C07207=1031.789,-57.070,-84.960,167.872,41.693,157.752
C07208=1031.783,-57.319,-84.950,167.870,41.694,157.752
C07209=1031.776,-57.569,-84.938,167.867,41.696,157.752
C07210=1031.770,-57.819,-84.925,167.864,41.697,157.752
C07211=1031.764,-58.068,-84.913,167.861,41.698,157.752
C07212=1031.758,-58.318,-84.902,167.859,41.700,157.752
C07213=1031.751,-58.567,-84.890,167.857,41.701,157.752
C07214=1031.746,-58.817,-84.878,167.854,41.702,157.752
C07215=1031.740,-59.067,-84.867,167.851,41.703,157.752
C07216=1031.733,-59.316,-84.855,167.848,41.705,157.752
C07217=1031.726,-59.566,-84.843,167.845,41.706,157.752
C07218=1031.721,-59.816,-84.830,167.842,41.707,157.752
C07219=1031.715,-60.065,-84.820,167.840,41.709,157.752
C07220=1031.708,-60.315,-84.808,167.838,41.710,157.752
C07221=1031.702,-60.564,-84.796,167.835,41.711,157.753
C07222=1031.697,-60.814,-84.784,167.832,41.712,157.753
C07223=1031.690,-61.064,-84.772,167.829,41.713,157.753
C07224=1031.683,-61.313,-84.760,167.826,41.714,157.753
C07225=1031.678,-61.563,-84.749,167.824,41.716,157.753
C07226=1031.672,-61.813,-84.737,167.821,41.717,157.753
C07227=1031.665,-62.063,-84.726,167.818,41.718,157.753
C07228=1031.659,-62.312,-84.714,167.815,41.719,157.753
C07229=1031.653,-62.561,-84.702,167.813,41.720,157.753
C07230=1031.647,-62.812,-84.690,167.811,41.722,157.753
C07231=1031.641,-63.061,-84.679,167.808,41.723,157.753
C07232=1031.635,-63.311,-84.667,167.805,41.724,157.753
C07233=1031.628,-63.560,-84.655,167.802,41.726,157.753
C07234=1031.623,-63.810,-84.644,167.799,41.727,157.753
C07235=1031.616,-64.060,-84.632,167.796,41.728,157.753
C07236=1031.610,-64.309,-84.620,167.793,41.729,157.753
C07237=1031.604,-64.559,-84.609,167.791,41.731,157.753
C07238=1031.597,-64.808,-84.597,167.789,41.732,157.753
C07239=1031.592,-65.058,-84.586,167.786,41.733,157.754
C07240=1031.586,-65.308,-84.574,167.783,41.735,157.754
C07241=1031.580,-65.557,-84.563,167.780,41.736,157.754
C07242=1031.573,-65.807,-84.551,167.778,41.737,157.754
C07243=1031.568,-66.057,-84.539,167.775,41.738,157.754
C07244=1031.562,-66.306,-84.527,167.772,41.740,157.754
C07245=1031.555,-66.556,-84.516,167.769,41.741,157.754
C07246=1031.549,-66.806,-84.505,167.766,41.742,157.754
C07247=1031.543,-67.055,-84.493,167.764,41.744,157.754
C07248=1031.538,-67.305,-84.482,167.762,41.744,157.754
C07249=1031.531,-67.555,-84.470,167.759,41.746,157.754
C07250=1031.525,-67.804,-84.459,167.756,41.747,157.754
C07251=1031.519,-68.087,-84.446,167.753,41.748,157.754
C07252=1031.512,-68.370,-84.433,167.749,41.750,157.754
C07253=1031.505,-68.652,-84.419,167.747,41.751,157.754
C07254=1031.498,-68.934,-84.406,167.744,41.752,157.754
C07255=1031.492,-69.185,-84.395,167.741,41.753,157.754
C07256=1031.486,-69.434,-84.384,167.738,41.755,157.755
C07257=1031.479,-69.684,-84.372,167.735,41.756,157.755
C07258=1031.474,-69.933,-84.361,167.732,41.757,157.755
C07259=1031.467,-70.183,-84.350,167.730,41.759,157.755
C07260=1031.462,-70.432,-84.338,167.727,41.760,157.755
C07261=1031.456,-70.682,-84.327,167.724,41.761,157.755
C07262=1031.450,-70.932,-84.316,167.721,41.762,157.755
C07263=1031.444,-71.181,-84.304,167.719,41.764,157.755
C07264=1031.438,-71.431,-84.293,167.717,41.765,157.755
C07265=1031.433,-71.681,-84.281,167.714,41.766,157.755
C07266=1031.426,-71.931,-84.270,167.711,41.767,157.755
C07267=1031.420,-72.180,-84.259,167.708,41.769,157.755
C07268=1031.414,-72.430,-84.247,167.705,41.770,157.755
C07269=1031.408,-72.680,-84.237,167.702,41.771,157.755
C07270=1031.402,-72.929,-84.225,167.700,41.773,157.755
C07271=1031.396,-73.179,-84.213,167.697,41.774,157.755
C07272=1031.391,-73.429,-84.202,167.694,41.775,157.755
C07273=1031.384,-73.679,-84.191,167.691,41.776,157.755
C07274=1031.378,-73.928,-84.179,167.689,41.778,157.755
///RCONF 1,0,0,1,0,0,0,0,0,0,0,0,0,0,0,0,0,0,0,0,0,0,0,0
C07275=1031.373,-74.177,-84.169,167.686,41.779,157.755
C07276=1031.366,-74.427,-84.157,167.684,41.780,157.756
C07277=1031.361,-74.677,-84.146,167.681,41.781,157.756
C07278=1031.354,-74.927,-84.135,167.678,41.783,157.756
C07279=1031.348,-75.177,-84.124,167.675,41.784,157.756
C07280=1031.343,-75.426,-84.113,167.672,41.785,157.756
C07281=1031.336,-75.676,-84.103,167.670,41.787,157.756
C07282=1031.330,-75.925,-84.092,167.667,41.788,157.756
C07283=1031.324,-76.176,-84.081,167.664,41.790,157.756
C07284=1031.318,-76.424,-84.069,167.661,41.791,157.756
C07285=1031.312,-76.674,-84.058,167.658,41.793,157.756
C07286=1031.305,-76.924,-84.047,167.656,41.794,157.756
C07287=1031.300,-77.174,-84.036,167.653,41.796,157.756
C07288=1031.294,-77.423,-84.025,167.650,41.797,157.756
C07289=1031.287,-77.673,-84.015,167.647,41.798,157.757
C07290=1031.281,-77.922,-84.004,167.644,41.799,157.757
C07291=1031.275,-78.172,-83.993,167.642,41.801,157.757
C07292=1031.269,-78.422,-83.982,167.639,41.802,157.757
C07293=1031.263,-78.672,-83.971,167.636,41.803,157.757
C07294=1031.258,-78.921,-83.960,167.633,41.805,157.757
C07295=1031.251,-79.171,-83.949,167.630,41.806,157.757
C07296=1031.246,-79.421,-83.938,167.628,41.808,157.757
C07297=1031.239,-79.670,-83.927,167.625,41.809,157.757
C07298=1031.233,-79.920,-83.916,167.622,41.811,157.757
C07299=1031.227,-80.170,-83.906,167.619,41.812,157.757
C07300=1031.222,-80.420,-83.895,167.617,41.814,157.757
C07301=1031.214,-80.670,-83.884,167.614,41.815,157.757
C07302=1031.209,-80.919,-83.874,167.611,41.816,157.757
C07303=1031.202,-81.168,-83.863,167.608,41.818,157.758
C07304=1031.196,-81.418,-83.852,167.606,41.820,157.758
C07305=1031.190,-81.669,-83.842,167.603,41.821,157.758
C07306=1031.184,-81.918,-83.832,167.600,41.823,157.758
C07307=1031.178,-82.167,-83.821,167.597,41.825,157.758
C07308=1031.171,-82.417,-83.810,167.594,41.826,157.758
C07309=1031.165,-82.667,-83.799,167.592,41.827,157.758
C07310=1031.160,-82.917,-83.789,167.589,41.828,157.758
C07311=1031.153,-83.166,-83.779,167.586,41.830,157.758
C07312=1031.147,-83.416,-83.767,167.582,41.832,157.758
C07313=1031.141,-83.666,-83.757,167.580,41.833,157.758
C07314=1031.135,-83.915,-83.747,167.577,41.835,157.759
C07315=1031.128,-84.199,-83.734,167.574,41.837,157.759
C07316=1031.121,-84.485,-83.722,167.570,41.839,157.759
C07317=1031.114,-84.769,-83.710,167.568,41.840,157.759
C07318=1031.107,-85.054,-83.698,167.564,41.842,157.759
C07319=1031.101,-85.303,-83.688,167.561,41.843,157.759
C07320=1031.096,-85.553,-83.678,167.558,41.845,157.759
C07321=1031.089,-85.803,-83.667,167.556,41.847,157.759
C07322=1031.083,-86.053,-83.656,167.553,41.848,157.759
C07323=1031.077,-86.303,-83.646,167.550,41.850,157.760
C07324=1031.071,-86.552,-83.636,167.547,41.851,157.760
C07325=1031.065,-86.802,-83.626,167.545,41.852,157.760
C07326=1031.059,-87.051,-83.615,167.542,41.854,157.760
C07327=1031.053,-87.302,-83.604,167.539,41.855,157.760
C07328=1031.046,-87.551,-83.595,167.536,41.857,157.760
C07329=1031.041,-87.801,-83.584,167.534,41.859,157.760
C07330=1031.035,-88.050,-83.573,167.531,41.860,157.760
C07331=1031.029,-88.300,-83.563,167.528,41.862,157.760
C07332=1031.023,-88.550,-83.552,167.525,41.863,157.760
C07333=1031.017,-88.799,-83.543,167.522,41.865,157.760
C07334=1031.010,-89.050,-83.532,167.520,41.866,157.761
C07335=1031.004,-89.299,-83.522,167.517,41.868,157.761
C07336=1030.999,-89.549,-83.511,167.514,41.869,157.761
///RCONF 1,0,0,0,0,0,0,0,0,0,0,0,0,0,0,0,0,0,0,0,0,0,0,0
C07337=1030.992,-89.798,-83.501,167.510,41.871,157.761
C07338=1030.987,-90.048,-83.491,167.508,41.873,157.761
C07339=1030.981,-90.298,-83.480,167.505,41.874,157.761
C07340=1030.975,-90.547,-83.470,167.502,41.876,157.761
C07341=1030.969,-90.797,-83.459,167.499,41.877,157.761
C07342=1030.963,-91.047,-83.450,167.496,41.878,157.761
C07343=1030.957,-91.296,-83.439,167.494,41.880,157.761
C07344=1030.951,-91.546,-83.429,167.491,41.882,157.761
C07345=1030.945,-91.796,-83.418,167.488,41.883,157.761
C07346=1030.938,-92.046,-83.409,167.485,41.885,157.762
C07347=1030.933,-92.296,-83.398,167.483,41.887,157.762
C07348=1030.926,-92.545,-83.388,167.480,41.888,157.762
C07349=1030.921,-92.795,-83.378,167.477,41.889,157.762
C07350=1030.915,-93.045,-83.368,167.475,41.891,157.762
C07351=1030.909,-93.295,-83.357,167.472,41.892,157.762
C07352=1030.903,-93.544,-83.347,167.469,41.894,157.762
C07353=1030.897,-93.794,-83.337,167.466,41.895,157.762
C07354=1030.892,-94.044,-83.327,167.463,41.897,157.762
C07355=1030.885,-94.293,-83.317,167.460,41.899,157.762
C07356=1030.880,-94.543,-83.306,167.457,41.900,157.762
C07357=1030.873,-94.793,-83.296,167.454,41.902,157.763
C07358=1030.868,-95.043,-83.286,167.451,41.903,157.763
C07359=1030.862,-95.292,-83.276,167.448,41.904,157.763
C07360=1030.856,-95.542,-83.266,167.446,41.906,157.763
C07361=1030.850,-95.792,-83.256,167.443,41.908,157.763
C07362=1030.844,-96.042,-83.246,167.440,41.909,157.763
C07363=1030.839,-96.290,-83.236,167.437,41.911,157.763
C07364=1030.833,-96.540,-83.226,167.435,41.913,157.763
C07365=1030.827,-96.790,-83.216,167.432,41.914,157.763
C07366=1030.821,-97.040,-83.205,167.429,41.915,157.763
C07367=1030.815,-97.290,-83.196,167.426,41.917,157.764
C07368=1030.810,-97.540,-83.186,167.424,41.918,157.764
C07369=1030.803,-97.789,-83.176,167.421,41.920,157.764
C07370=1030.797,-98.039,-83.166,167.417,41.922,157.764
C07371=1030.792,-98.289,-83.156,167.414,41.924,157.764
C07372=1030.785,-98.539,-83.146,167.412,41.925,157.764
C07373=1030.779,-98.788,-83.136,167.409,41.927,157.764
C07374=1030.773,-99.038,-83.127,167.406,41.929,157.764
C07375=1030.768,-99.288,-83.117,167.404,41.930,157.764
C07376=1030.761,-99.538,-83.107,167.401,41.932,157.764
C07377=1030.755,-99.787,-83.097,167.398,41.934,157.765
C07378=1030.749,-100.037,-83.087,167.394,41.936,157.765
C07379=1030.743,-100.324,-83.076,167.392,41.937,157.765
C07380=1030.736,-100.611,-83.065,167.388,41.939,157.765
C07381=1030.729,-100.898,-83.054,167.385,41.941,157.765
C07382=1030.722,-101.184,-83.043,167.382,41.943,157.765
C07383=1030.716,-101.434,-83.033,167.379,41.945,157.765
C07384=1030.710,-101.684,-83.023,167.376,41.946,157.765
C07385=1030.704,-101.934,-83.014,167.373,41.948,157.766
C07386=1030.698,-102.184,-83.004,167.371,41.950,157.766
C07387=1030.693,-102.433,-82.995,167.367,41.952,157.766
C07388=1030.686,-102.683,-82.985,167.364,41.954,157.766
C07389=1030.681,-102.933,-82.975,167.361,41.955,157.766
C07390=1030.674,-103.182,-82.965,167.359,41.956,157.766
C07391=1030.668,-103.432,-82.955,167.356,41.958,157.766
C07392=1030.662,-103.682,-82.946,167.353,41.960,157.766
C07393=1030.657,-103.931,-82.937,167.351,41.962,157.766
C07394=1030.651,-104.182,-82.927,167.348,41.964,157.767
C07395=1030.645,-104.431,-82.917,167.344,41.965,157.767
C07396=1030.639,-104.681,-82.908,167.341,41.967,157.767
C07397=1030.633,-104.931,-82.898,167.339,41.968,157.767
C07398=1030.627,-105.180,-82.889,167.336,41.970,157.767
C07399=1030.622,-105.430,-82.879,167.333,41.972,157.767
C07400=1030.616,-105.680,-82.869,167.330,41.974,157.767
C07401=1030.610,-105.930,-82.860,167.328,41.975,157.767
C07402=1030.603,-106.180,-82.850,167.325,41.977,157.767
C07403=1030.598,-106.429,-82.841,167.321,41.979,157.768
C07404=1030.592,-106.678,-82.831,167.319,41.981,157.768
C07405=1030.586,-106.929,-82.821,167.316,41.983,157.768
C07406=1030.580,-107.179,-82.812,167.313,41.984,157.768
C07407=1030.575,-107.428,-82.803,167.310,41.985,157.768
C07408=1030.569,-107.678,-82.794,167.308,41.987,157.768
C07409=1030.562,-107.928,-82.784,167.305,41.989,157.768
C07410=1030.556,-108.177,-82.775,167.301,41.991,157.768
C07411=1030.551,-108.427,-82.765,167.299,41.993,157.768
C07412=1030.545,-108.677,-82.756,167.296,41.995,157.769
C07413=1030.539,-108.927,-82.747,167.293,41.996,157.769
C07414=1030.533,-109.176,-82.738,167.290,41.998,157.769
C07415=1030.527,-109.426,-82.728,167.288,42.000,157.769
C07416=1030.521,-109.676,-82.719,167.284,42.002,157.769
C07417=1030.515,-109.926,-82.710,167.281,42.004,157.769
C07418=1030.509,-110.175,-82.700,167.279,42.005,157.769
C07419=1030.503,-110.425,-82.691,167.276,42.008,157.770
C07420=1030.497,-110.675,-82.682,167.273,42.010,157.770
C07421=1030.492,-110.924,-82.673,167.270,42.011,157.770
C07422=1030.486,-111.174,-82.663,167.267,42.013,157.770
C07423=1030.480,-111.425,-82.654,167.264,42.015,157.770
C07424=1030.474,-111.674,-82.645,167.262,42.017,157.770
C07425=1030.468,-111.923,-82.636,167.259,42.019,157.770
C07426=1030.462,-112.174,-82.627,167.256,42.020,157.770
C07427=1030.457,-112.423,-82.618,167.252,42.022,157.771
C07428=1030.450,-112.673,-82.608,167.250,42.024,157.771
C07429=1030.444,-112.923,-82.599,167.247,42.026,157.771
C07430=1030.439,-113.172,-82.590,167.244,42.028,157.771
C07431=1030.433,-113.422,-82.580,167.242,42.029,157.771
C07432=1030.427,-113.672,-82.572,167.239,42.031,157.771
C07433=1030.421,-113.922,-82.562,167.235,42.033,157.771
C07434=1030.415,-114.172,-82.554,167.233,42.035,157.771
C07435=1030.410,-114.421,-82.544,167.230,42.037,157.772
C07436=1030.404,-114.671,-82.535,167.227,42.038,157.772
C07437=1030.398,-114.920,-82.527,167.224,42.040,157.772
C07438=1030.392,-115.170,-82.517,167.222,42.042,157.772
C07439=1030.386,-115.420,-82.508,167.218,42.044,157.772
C07440=1030.380,-115.670,-82.499,167.215,42.046,157.772
C07441=1030.374,-115.920,-82.490,167.213,42.047,157.772
C07442=1030.369,-116.169,-82.481,167.210,42.050,157.772
C07443=1030.361,-116.456,-82.472,167.206,42.052,157.773
C07444=1030.355,-116.743,-82.461,167.203,42.054,157.773
C07445=1030.348,-117.028,-82.451,167.200,42.056,157.773
C07446=1030.342,-117.315,-82.441,167.196,42.058,157.773
C07447=1030.336,-117.565,-82.432,167.194,42.060,157.773
C07448=1030.330,-117.815,-82.423,167.191,42.062,157.773
C07449=1030.325,-118.064,-82.413,167.188,42.064,157.774
C07450=1030.318,-118.314,-82.405,167.185,42.066,157.774
C07451=1030.312,-118.563,-82.396,167.182,42.068,157.774
C07452=1030.306,-118.814,-82.387,167.179,42.070,157.774
C07453=1030.301,-119.064,-82.378,167.177,42.071,157.774
C07454=1030.294,-119.313,-82.370,167.174,42.073,157.774
C07455=1030.288,-119.563,-82.361,167.170,42.075,157.774
C07456=1030.283,-119.813,-82.352,167.168,42.078,157.774
C07457=1030.277,-120.063,-82.343,167.165,42.079,157.775
C07458=1030.272,-120.313,-82.334,167.162,42.081,157.775
C07459=1030.265,-120.561,-82.326,167.159,42.083,157.775
C07460=1030.260,-120.812,-82.317,167.156,42.085,157.775
C07461=1030.254,-121.061,-82.308,167.153,42.087,157.775
C07462=1030.248,-121.312,-82.300,167.151,42.089,157.775
C07463=1030.242,-121.561,-82.291,167.148,42.091,157.775
C07464=1030.236,-121.811,-82.282,167.144,42.093,157.776
C07465=1030.231,-122.061,-82.274,167.142,42.095,157.776
C07466=1030.225,-122.311,-82.264,167.139,42.096,157.776
C07467=1030.219,-122.560,-82.256,167.136,42.099,157.776
C07468=1030.213,-122.810,-82.247,167.134,42.101,157.776
C07469=1030.208,-123.060,-82.239,167.130,42.103,157.776
C07470=1030.202,-123.309,-82.230,167.127,42.104,157.776
C07471=1030.196,-123.559,-82.221,167.124,42.106,157.777
C07472=1030.190,-123.809,-82.213,167.122,42.108,157.777
C07473=1030.184,-124.059,-82.204,167.119,42.110,157.777
C07474=1030.179,-124.309,-82.196,167.116,42.112,157.777
C07475=1030.173,-124.558,-82.187,167.113,42.114,157.777
C07476=1030.167,-124.808,-82.178,167.110,42.116,157.777
C07477=1030.161,-125.058,-82.170,167.108,42.118,157.777
C07478=1030.155,-125.308,-82.161,167.104,42.120,157.778
C07479=1030.150,-125.558,-82.153,167.101,42.122,157.778
C07480=1030.144,-125.807,-82.145,167.098,42.124,157.778
C07481=1030.138,-126.058,-82.136,167.096,42.126,157.778
C07482=1030.132,-126.307,-82.128,167.092,42.128,157.778
C07483=1030.126,-126.556,-82.119,167.090,42.130,157.778
C07484=1030.121,-126.807,-82.110,167.087,42.133,157.779
C07485=1030.115,-127.056,-82.102,167.084,42.134,157.779
C07486=1030.109,-127.306,-82.093,167.082,42.136,157.779
C07487=1030.103,-127.556,-82.086,167.078,42.139,157.779
C07488=1030.097,-127.806,-82.077,167.075,42.140,157.779
C07489=1030.092,-128.055,-82.068,167.073,42.142,157.779
C07490=1030.087,-128.305,-82.059,167.070,42.143,157.779
C07491=1030.082,-128.554,-82.049,167.067,42.144,157.779
C07492=1030.080,-128.803,-82.038,167.065,42.145,157.779
C07493=1030.076,-129.053,-82.027,167.063,42.144,157.779
C07494=1030.074,-129.303,-82.016,167.059,42.144,157.779
C07495=1030.072,-129.554,-82.004,167.058,42.143,157.778
C07496=1030.071,-129.803,-81.991,167.056,42.142,157.778
C07497=1030.071,-130.053,-81.978,167.053,42.139,157.777
C07498=1030.071,-130.303,-81.964,167.051,42.137,157.777
C07499=1030.071,-130.553,-81.950,167.049,42.134,157.776
C07500=1030.073,-130.803,-81.934,167.048,42.131,157.776
C07501=1030.075,-131.053,-81.918,167.045,42.127,157.775
C07502=1030.077,-131.302,-81.902,167.044,42.123,157.774
C07503=1030.081,-131.553,-81.885,167.043,42.118,157.773
C07504=1030.085,-131.803,-81.868,167.042,42.112,157.772
C07505=1030.089,-132.053,-81.850,167.040,42.107,157.771
C07506=1030.095,-132.302,-81.831,167.039,42.101,157.770
C07507=1029.776,-132.327,-82.136,166.990,42.343,157.807
C07508=1029.771,-132.078,-82.154,166.992,42.349,157.808
C07509=1029.767,-131.828,-82.172,166.993,42.355,157.809
C07510=1029.762,-131.577,-82.190,166.994,42.360,157.811
C07511=1029.759,-131.327,-82.206,166.996,42.365,157.811
C07512=1029.756,-131.077,-82.223,166.997,42.369,157.812
C07513=1029.755,-130.827,-82.238,166.999,42.373,157.813
C07514=1029.753,-130.578,-82.253,167.001,42.376,157.814
C07515=1029.752,-130.328,-82.268,167.003,42.379,157.814
C07516=1029.752,-130.078,-82.282,167.004,42.382,157.815
C07517=1029.753,-129.828,-82.295,167.007,42.383,157.815
C07518=1029.754,-129.578,-82.308,167.009,42.385,157.816
C07519=1029.755,-129.328,-82.320,167.011,42.386,157.816
C07520=1029.758,-129.079,-82.332,167.013,42.387,157.816
C07521=1029.760,-128.829,-82.343,167.016,42.386,157.816
C07522=1029.764,-128.579,-82.354,167.018,42.386,157.816
C07523=1029.769,-128.330,-82.364,167.021,42.386,157.817
C07524=1029.773,-128.080,-82.373,167.024,42.384,157.816
C07525=1029.778,-127.830,-82.381,167.027,42.382,157.816
C07526=1029.784,-127.580,-82.390,167.029,42.380,157.816
C07527=1029.790,-127.332,-82.398,167.032,42.378,157.816
C07528=1029.795,-127.082,-82.407,167.036,42.376,157.816
C07529=1029.802,-126.832,-82.415,167.038,42.374,157.816
C07530=1029.807,-126.582,-82.424,167.041,42.372,157.816
C07531=1029.812,-126.332,-82.432,167.044,42.370,157.816
C07532=1029.819,-126.082,-82.440,167.047,42.368,157.815
C07533=1029.824,-125.833,-82.449,167.050,42.366,157.815
C07534=1029.830,-125.583,-82.457,167.053,42.364,157.815
C07535=1029.836,-125.333,-82.466,167.055,42.362,157.815
C07536=1029.841,-125.083,-82.474,167.059,42.360,157.815
C07537=1029.848,-124.833,-82.482,167.062,42.358,157.815
C07538=1029.854,-124.584,-82.492,167.064,42.355,157.814
C07539=1029.860,-124.334,-82.499,167.068,42.353,157.814
C07540=1029.865,-124.084,-82.508,167.070,42.352,157.814
C07541=1029.871,-123.834,-82.517,167.073,42.349,157.814
C07542=1029.877,-123.584,-82.526,167.076,42.347,157.814
C07543=1029.883,-123.335,-82.534,167.078,42.345,157.814
C07544=1029.888,-123.085,-82.543,167.082,42.344,157.814
C07545=1029.894,-122.835,-82.552,167.085,42.342,157.813
C07546=1029.900,-122.586,-82.559,167.087,42.339,157.813
C07547=1029.906,-122.335,-82.568,167.090,42.337,157.813
C07548=1029.911,-122.086,-82.578,167.094,42.335,157.813
C07549=1029.917,-121.836,-82.586,167.096,42.334,157.813
C07550=1029.923,-121.586,-82.594,167.099,42.331,157.813
C07551=1029.929,-121.337,-82.603,167.102,42.329,157.813
C07552=1029.935,-121.087,-82.612,167.105,42.327,157.812
C07553=1029.940,-120.837,-82.621,167.108,42.326,157.812
C07554=1029.947,-120.587,-82.629,167.110,42.323,157.812
C07555=1029.952,-120.338,-82.638,167.113,42.321,157.812
C07556=1029.958,-120.087,-82.647,167.116,42.320,157.812
C07557=1029.963,-119.838,-82.656,167.120,42.318,157.812
C07558=1029.970,-119.588,-82.665,167.122,42.316,157.812
C07559=1029.976,-119.338,-82.673,167.125,42.313,157.811
C07560=1029.981,-119.088,-82.682,167.127,42.311,157.811
C07561=1029.987,-118.839,-82.691,167.131,42.310,157.811
C07562=1029.993,-118.589,-82.700,167.134,42.308,157.811
C07563=1029.998,-118.339,-82.709,167.137,42.306,157.811
C07564=1030.005,-118.089,-82.717,167.139,42.303,157.811
C07565=1030.010,-117.840,-82.726,167.143,42.302,157.811
C07566=1030.016,-117.590,-82.735,167.145,42.300,157.810
C07567=1030.022,-117.340,-82.744,167.148,42.298,157.810
C07568=1030.029,-117.054,-82.754,167.152,42.295,157.810
C07569=1030.035,-116.768,-82.765,167.154,42.293,157.810
C07570=1030.042,-116.481,-82.774,167.158,42.292,157.810
C07571=1030.049,-116.195,-82.785,167.162,42.289,157.810
C07572=1030.055,-115.945,-82.794,167.164,42.287,157.810
C07573=1030.061,-115.695,-82.803,167.167,42.285,157.809
C07574=1030.066,-115.446,-82.812,167.170,42.284,157.809
C07575=1030.073,-115.196,-82.821,167.173,42.281,157.809
C07576=1030.078,-114.947,-82.830,167.176,42.279,157.809
C07577=1030.084,-114.696,-82.839,167.179,42.277,157.809
C07578=1030.090,-114.446,-82.848,167.181,42.275,157.809
C07579=1030.096,-114.197,-82.857,167.185,42.274,157.809
C07580=1030.102,-113.947,-82.866,167.188,42.272,157.809
C07581=1030.107,-113.697,-82.875,167.190,42.270,157.808
C07582=1030.113,-113.447,-82.884,167.193,42.268,157.808
C07583=1030.119,-113.198,-82.894,167.196,42.266,157.808
C07584=1030.125,-112.948,-82.902,167.199,42.265,157.808
C07585=1030.131,-112.698,-82.912,167.202,42.263,157.808
C07586=1030.136,-112.448,-82.920,167.205,42.260,157.808
C07587=1030.142,-112.199,-82.930,167.207,42.258,157.808
C07588=1030.148,-111.949,-82.940,167.210,42.257,157.807
C07589=1030.154,-111.699,-82.948,167.213,42.255,157.807
C07590=1030.160,-111.449,-82.958,167.217,42.253,157.807
C07591=1030.166,-111.199,-82.967,167.219,42.251,157.807
C07592=1030.171,-110.950,-82.976,167.222,42.249,157.807
C07593=1030.177,-110.700,-82.985,167.225,42.247,157.807
C07594=1030.184,-110.450,-82.995,167.227,42.246,157.807
C07595=1030.189,-110.200,-83.003,167.231,42.244,157.807
C07596=1030.195,-109.951,-83.013,167.234,42.242,157.807
C07597=1030.201,-109.701,-83.022,167.236,42.240,157.806
C07598=1030.207,-109.452,-83.032,167.239,42.238,157.806
C07599=1030.213,-109.201,-83.041,167.242,42.237,157.806
C07600=1030.219,-108.951,-83.050,167.246,42.235,157.806
C07601=1030.224,-108.702,-83.059,167.248,42.233,157.806
C07602=1030.231,-108.453,-83.069,167.251,42.230,157.806
C07603=1030.236,-108.202,-83.078,167.253,42.229,157.806
C07604=1030.243,-107.952,-83.087,167.256,42.227,157.805
C07605=1030.248,-107.703,-83.096,167.260,42.225,157.805
C07606=1030.254,-107.453,-83.106,167.263,42.223,157.805
C07607=1030.261,-107.204,-83.116,167.265,42.221,157.805
C07608=1030.266,-106.953,-83.124,167.268,42.219,157.805
C07609=1030.272,-106.704,-83.134,167.271,42.218,157.805
C07610=1030.278,-106.454,-83.143,167.273,42.216,157.805
C07611=1030.284,-106.204,-83.153,167.277,42.214,157.805
C07612=1030.290,-105.954,-83.163,167.280,42.213,157.805
C07613=1030.295,-105.705,-83.172,167.283,42.211,157.804
C07614=1030.302,-105.456,-83.182,167.285,42.209,157.804
C07615=1030.308,-105.206,-83.191,167.288,42.207,157.804
C07616=1030.314,-104.956,-83.201,167.291,42.206,157.804
C07617=1030.319,-104.705,-83.210,167.294,42.204,157.804
C07618=1030.325,-104.456,-83.220,167.297,42.202,157.804
C07619=1030.331,-104.206,-83.229,167.300,42.200,157.804
C07620=1030.337,-103.957,-83.239,167.302,42.198,157.804
C07621=1030.343,-103.707,-83.248,167.305,42.197,157.803
C07622=1030.348,-103.457,-83.258,167.308,42.195,157.803
C07623=1030.354,-103.208,-83.268,167.311,42.193,157.803
C07624=1030.360,-102.958,-83.277,167.314,42.191,157.803
C07625=1030.366,-102.708,-83.287,167.317,42.189,157.803
C07626=1030.373,-102.458,-83.296,167.320,42.188,157.803
C07627=1030.378,-102.208,-83.306,167.323,42.186,157.803
C07628=1030.384,-101.959,-83.316,167.325,42.185,157.803
C07629=1030.390,-101.709,-83.325,167.328,42.183,157.803
C07630=1030.396,-101.459,-83.335,167.332,42.181,157.803
C07631=1030.402,-101.210,-83.346,167.334,42.179,157.802
C07632=1030.408,-100.923,-83.357,167.337,42.177,157.802
C07633=1030.416,-100.636,-83.368,167.341,42.175,157.802
C07634=1030.422,-100.349,-83.379,167.344,42.173,157.802
C07635=1030.429,-100.063,-83.390,167.347,42.171,157.802
C07636=1030.435,-99.813,-83.399,167.350,42.169,157.802
C07637=1030.441,-99.563,-83.409,167.352,42.167,157.802
C07638=1030.447,-99.313,-83.419,167.356,42.165,157.802
C07639=1030.453,-99.063,-83.428,167.359,42.164,157.802
C07640=1030.460,-98.814,-83.439,167.362,42.163,157.801
C07641=1030.465,-98.564,-83.449,167.364,42.161,157.801
C07642=1030.471,-98.314,-83.458,167.367,42.159,157.801
C07643=1030.477,-98.064,-83.468,167.370,42.157,157.801
C07644=1030.483,-97.815,-83.478,167.373,42.155,157.801
C07645=1030.489,-97.564,-83.488,167.376,42.154,157.801
C07646=1030.495,-97.315,-83.498,167.379,42.152,157.801
C07647=1030.501,-97.065,-83.508,167.382,42.151,157.801
C07648=1030.506,-96.816,-83.517,167.384,42.149,157.800
C07649=1030.512,-96.566,-83.527,167.387,42.147,157.800
C07650=1030.518,-96.317,-83.538,167.390,42.146,157.800
C07651=1030.524,-96.067,-83.548,167.393,42.144,157.800
C07652=1030.530,-95.817,-83.557,167.395,42.142,157.800
C07653=1030.536,-95.567,-83.568,167.398,42.141,157.800
C07654=1030.542,-95.318,-83.578,167.401,42.140,157.800
C07655=1030.547,-95.067,-83.588,167.405,42.138,157.800
C07656=1030.554,-94.818,-83.598,167.407,42.136,157.800
C07657=1030.559,-94.568,-83.609,167.410,42.134,157.800
C07658=1030.565,-94.318,-83.618,167.413,42.133,157.800
C07659=1030.571,-94.069,-83.629,167.416,42.131,157.799
C07660=1030.577,-93.819,-83.639,167.418,42.129,157.799
C07661=1030.583,-93.570,-83.649,167.421,42.128,157.799
C07662=1030.589,-93.320,-83.659,167.424,42.127,157.799
C07663=1030.595,-93.070,-83.669,167.427,42.125,157.799
C07664=1030.601,-92.821,-83.679,167.429,42.123,157.799
C07665=1030.607,-92.570,-83.690,167.432,42.122,157.799
C07666=1030.612,-92.321,-83.700,167.436,42.120,157.799
C07667=1030.618,-92.071,-83.710,167.439,42.118,157.799
C07668=1030.624,-91.822,-83.721,167.441,42.117,157.799
C07669=1030.630,-91.572,-83.730,167.444,42.115,157.799
C07670=1030.636,-91.322,-83.741,167.447,42.113,157.798
C07671=1030.642,-91.073,-83.751,167.449,42.112,157.798
C07672=1030.648,-90.822,-83.761,167.452,42.111,157.798
C07673=1030.654,-90.573,-83.771,167.455,42.109,157.798
C07674=1030.660,-90.322,-83.782,167.458,42.107,157.798
C07675=1030.667,-90.073,-83.792,167.461,42.106,157.798
C07676=1030.672,-89.823,-83.802,167.463,42.104,157.798
C07677=1030.679,-89.574,-83.813,167.466,42.102,157.798
C07678=1030.684,-89.324,-83.824,167.470,42.100,157.798
C07679=1030.690,-89.074,-83.834,167.473,42.099,157.798
C07680=1030.696,-88.825,-83.844,167.475,42.098,157.798
C07681=1030.702,-88.575,-83.854,167.478,42.096,157.797
C07682=1030.708,-88.326,-83.864,167.481,42.095,157.797
C07683=1030.714,-88.076,-83.875,167.484,42.093,157.797
C07684=1030.721,-87.826,-83.885,167.486,42.091,157.797
C07685=1030.726,-87.576,-83.896,167.489,42.089,157.797
C07686=1030.732,-87.326,-83.906,167.492,42.088,157.797
C07687=1030.738,-87.077,-83.917,167.495,42.087,157.797
C07688=1030.744,-86.827,-83.927,167.497,42.085,157.797
C07689=1030.750,-86.578,-83.937,167.500,42.084,157.797
C07690=1030.757,-86.328,-83.948,167.503,42.082,157.797
C07691=1030.763,-86.078,-83.958,167.507,42.080,157.797
C07692=1030.768,-85.828,-83.969,167.509,42.079,157.797
C07693=1030.774,-85.579,-83.980,167.512,42.077,157.796
C07694=1030.780,-85.329,-83.989,167.515,42.075,157.796
C07695=1030.786,-85.080,-84.000,167.517,42.074,157.796
C07696=1030.793,-84.794,-84.012,167.520,42.072,157.796
C07697=1030.801,-84.510,-84.024,167.524,42.070,157.796
C07698=1030.808,-84.225,-84.036,167.527,42.069,157.796
C07699=1030.814,-83.941,-84.047,167.530,42.067,157.796
C07700=1030.820,-83.691,-84.058,167.533,42.065,157.796
C07701=1030.827,-83.442,-84.069,167.536,42.063,157.796
C07702=1030.833,-83.192,-84.080,167.539,42.062,157.795
C07703=1030.838,-82.942,-84.090,167.541,42.060,157.795
C07704=1030.845,-82.692,-84.100,167.544,42.059,157.795
C07705=1030.851,-82.443,-84.111,167.547,42.057,157.795
C07706=1030.858,-82.193,-84.122,167.550,42.056,157.795
C07707=1030.863,-81.943,-84.132,167.552,42.054,157.795
C07708=1030.869,-81.694,-84.143,167.556,42.052,157.795
C07709=1030.876,-81.444,-84.154,167.559,42.050,157.795
C07710=1030.882,-81.194,-84.164,167.562,42.049,157.795
C07711=1030.888,-80.945,-84.175,167.564,42.047,157.795
C07712=1030.894,-80.695,-84.185,167.567,42.046,157.794
C07713=1030.900,-80.445,-84.196,167.570,42.045,157.794
C07714=1030.906,-80.195,-84.206,167.573,42.043,157.794
C07715=1030.912,-79.946,-84.217,167.575,42.041,157.794
C07716=1030.918,-79.696,-84.229,167.578,42.040,157.794
C07717=1030.924,-79.446,-84.239,167.581,42.038,157.794
C07718=1030.931,-79.197,-84.250,167.584,42.037,157.794
C07719=1030.937,-78.947,-84.261,167.586,42.035,157.794
C07720=1030.943,-78.697,-84.272,167.589,42.034,157.794
C07721=1030.948,-78.448,-84.283,167.592,42.032,157.794
C07722=1030.955,-78.198,-84.294,167.595,42.031,157.794
C07723=1030.961,-77.948,-84.305,167.598,42.030,157.794
C07724=1030.966,-77.699,-84.316,167.600,42.028,157.793
C07725=1030.973,-77.449,-84.327,167.603,42.027,157.793
C07726=1030.979,-77.199,-84.337,167.606,42.025,157.793
C07727=1030.985,-76.950,-84.348,167.609,42.024,157.793
C07728=1030.991,-76.700,-84.359,167.611,42.022,157.793
C07729=1030.997,-76.450,-84.370,167.614,42.021,157.793
C07730=1031.003,-76.201,-84.381,167.617,42.019,157.793
C07731=1031.009,-75.951,-84.392,167.620,42.018,157.793
C07732=1031.015,-75.701,-84.403,167.623,42.016,157.793
C07733=1031.020,-75.452,-84.414,167.625,42.015,157.793
C07734=1031.028,-75.202,-84.425,167.628,42.014,157.793
C07735=1031.033,-74.952,-84.436,167.631,42.012,157.793
C07736=1031.040,-74.702,-84.447,167.634,42.011,157.793
C07737=1031.045,-74.453,-84.458,167.637,42.010,157.793
C07738=1031.051,-74.203,-84.469,167.639,42.008,157.792
C07739=1031.058,-73.953,-84.481,167.642,42.007,157.792
C07740=1031.064,-73.704,-84.491,167.645,42.005,157.792
///RCONF 1,0,0,1,0,0,0,0,0,0,0,0,0,0,0,0,0,0,0,0,0,0,0,0
C07741=1031.070,-73.454,-84.503,167.648,42.004,157.792
C07742=1031.075,-73.204,-84.514,167.651,42.003,157.792
C07743=1031.081,-72.955,-84.525,167.653,42.001,157.792
C07744=1031.087,-72.705,-84.537,167.656,42.000,157.792
C07745=1031.093,-72.455,-84.548,167.659,41.999,157.792
C07746=1031.099,-72.205,-84.559,167.662,41.997,157.792
C07747=1031.105,-71.956,-84.570,167.665,41.996,157.792
C07748=1031.110,-71.707,-84.582,167.668,41.995,157.792
C07749=1031.117,-71.456,-84.593,167.670,41.993,157.792
C07750=1031.122,-71.207,-84.604,167.672,41.992,157.792
C07751=1031.129,-70.957,-84.616,167.675,41.991,157.792
C07752=1031.135,-70.708,-84.627,167.678,41.989,157.792
C07753=1031.141,-70.458,-84.638,167.681,41.988,157.792
C07754=1031.146,-70.208,-84.651,167.683,41.987,157.792
C07755=1031.153,-69.958,-84.662,167.686,41.985,157.791
C07756=1031.159,-69.709,-84.673,167.689,41.984,157.791
C07757=1031.165,-69.460,-84.684,167.692,41.983,157.791
C07758=1031.171,-69.210,-84.696,167.695,41.981,157.791
C07759=1031.176,-68.960,-84.707,167.697,41.980,157.791
C07760=1031.183,-68.678,-84.719,167.700,41.979,157.791
C07761=1031.190,-68.395,-84.732,167.703,41.978,157.791
C07762=1031.197,-68.113,-84.746,167.707,41.976,157.791
C07763=1031.204,-67.830,-84.759,167.710,41.975,157.791
C07764=1031.210,-67.580,-84.770,167.712,41.973,157.791
C07765=1031.216,-67.330,-84.781,167.715,41.972,157.791
C07766=1031.222,-67.081,-84.794,167.718,41.971,157.791
C07767=1031.228,-66.831,-84.805,167.721,41.969,157.791
C07768=1031.234,-66.582,-84.817,167.724,41.968,157.791
C07769=1031.240,-66.332,-84.828,167.726,41.967,157.791
C07770=1031.247,-66.082,-84.839,167.729,41.965,157.791
C07771=1031.252,-65.833,-84.851,167.732,41.964,157.791
C07772=1031.258,-65.583,-84.863,167.734,41.963,157.791
C07773=1031.265,-65.333,-84.874,167.737,41.961,157.790
C07774=1031.271,-65.084,-84.886,167.739,41.960,157.790
C07775=1031.277,-64.834,-84.897,167.742,41.959,157.790
C07776=1031.282,-64.585,-84.909,167.745,41.957,157.790
C07777=1031.289,-64.334,-84.920,167.748,41.956,157.790
C07778=1031.295,-64.086,-84.932,167.751,41.954,157.790
C07779=1031.301,-63.835,-84.943,167.753,41.953,157.790
C07780=1031.307,-63.586,-84.956,167.756,41.952,157.790
C07781=1031.313,-63.336,-84.967,167.759,41.950,157.790
C07782=1031.319,-63.086,-84.979,167.762,41.949,157.790
C07783=1031.326,-62.836,-84.990,167.765,41.948,157.790
C07784=1031.331,-62.587,-85.002,167.766,41.947,157.790
C07785=1031.338,-62.338,-85.014,167.769,41.946,157.790
C07786=1031.343,-62.088,-85.025,167.772,41.944,157.790
C07787=1031.350,-61.838,-85.037,167.775,41.943,157.790
C07788=1031.356,-61.588,-85.048,167.778,41.942,157.790
C07789=1031.362,-61.339,-85.060,167.781,41.941,157.790
C07790=1031.368,-61.090,-85.072,167.783,41.939,157.789
C07791=1031.375,-60.839,-85.083,167.786,41.938,157.789
C07792=1031.381,-60.590,-85.095,167.789,41.936,157.789
C07793=1031.387,-60.341,-85.108,167.792,41.935,157.789
C07794=1031.393,-60.090,-85.119,167.795,41.934,157.789
C07795=1031.399,-59.842,-85.130,167.797,41.932,157.789
C07796=1031.406,-59.592,-85.142,167.799,41.931,157.789
C07797=1031.411,-59.341,-85.154,167.802,41.930,157.789
C07798=1031.418,-59.092,-85.166,167.805,41.928,157.789
C07799=1031.424,-58.843,-85.178,167.808,41.927,157.789
C07800=1031.430,-58.593,-85.189,167.811,41.926,157.789
C07801=1031.436,-58.343,-85.202,167.813,41.924,157.789
C07802=1031.443,-58.093,-85.214,167.816,41.923,157.789
C07803=1031.449,-57.844,-85.225,167.819,41.922,157.789
C07804=1031.455,-57.594,-85.237,167.822,41.920,157.789
C07805=1031.461,-57.344,-85.249,167.825,41.919,157.789
C07806=1031.468,-57.095,-85.261,167.827,41.918,157.788
C07807=1031.474,-56.846,-85.273,167.829,41.917,157.788
///RCONF 1,0,0,0,0,0,0,0,0,0,0,0,0,0,0,0,0,0,0,0,0,0,0,0
C07808=1031.480,-56.595,-85.284,167.832,41.915,157.788
C07809=1031.486,-56.346,-85.296,167.835,41.914,157.788
C07810=1031.493,-56.096,-85.308,167.838,41.913,157.788
C07811=1031.499,-55.847,-85.320,167.840,41.912,157.788
C07812=1031.505,-55.598,-85.332,167.843,41.910,157.788
C07813=1031.511,-55.347,-85.344,167.846,41.909,157.788
C07814=1031.518,-55.098,-85.356,167.849,41.907,157.788
C07815=1031.524,-54.848,-85.368,167.852,41.906,157.788
C07816=1031.530,-54.599,-85.380,167.854,41.905,157.788
C07817=1031.536,-54.349,-85.392,167.856,41.903,157.788
C07818=1031.543,-54.100,-85.404,167.859,41.902,157.788
C07819=1031.549,-53.849,-85.416,167.862,41.901,157.788
C07820=1031.555,-53.600,-85.427,167.865,41.899,157.787
C07821=1031.562,-53.350,-85.439,167.867,41.898,157.787
C07822=1031.567,-53.101,-85.452,167.870,41.896,157.787
C07823=1031.574,-52.852,-85.464,167.873,41.895,157.787
C07824=1031.581,-52.569,-85.477,167.876,41.894,157.787
C07825=1031.588,-52.289,-85.491,167.879,41.893,157.787
C07826=1031.595,-52.007,-85.504,167.882,41.891,157.787
C07827=1031.603,-51.727,-85.518,167.885,41.890,157.787
C07828=1031.609,-51.477,-85.531,167.888,41.888,157.787
C07829=1031.615,-51.227,-85.542,167.891,41.887,157.787
C07830=1031.622,-50.978,-85.554,167.894,41.886,157.787
C07831=1031.628,-50.727,-85.566,167.895,41.884,157.787
C07832=1031.634,-50.478,-85.578,167.898,41.883,157.787
C07833=1031.640,-50.229,-85.591,167.901,41.882,157.787
C07834=1031.647,-49.979,-85.603,167.904,41.881,157.787
C07835=1031.653,-49.730,-85.616,167.907,41.880,157.787
C07836=1031.658,-49.480,-85.628,167.909,41.879,157.787
C07837=1031.664,-49.230,-85.641,167.911,41.877,157.786
C07838=1031.671,-48.980,-85.653,167.914,41.876,157.786
C07839=1031.677,-48.730,-85.665,167.917,41.875,157.786
C07840=1031.683,-48.480,-85.678,167.920,41.874,157.786
C07841=1031.689,-48.232,-85.689,167.923,41.873,157.786
C07842=1031.695,-47.982,-85.703,167.925,41.872,157.786
C07843=1031.701,-47.732,-85.715,167.928,41.871,157.786
C07844=1031.708,-47.483,-85.727,167.930,41.869,157.786
C07845=1031.714,-47.233,-85.740,167.933,41.868,157.786
C07846=1031.719,-46.983,-85.752,167.936,41.867,157.786
C07847=1031.726,-46.733,-85.764,167.938,41.866,157.786
C07848=1031.732,-46.484,-85.778,167.941,41.865,157.786
C07849=1031.738,-46.234,-85.790,167.944,41.864,157.786
C07850=1031.745,-45.985,-85.802,167.947,41.863,157.786
C07851=1031.751,-45.735,-85.815,167.949,41.861,157.786
C07852=1031.757,-45.486,-85.828,167.951,41.860,157.786
C07853=1031.764,-45.236,-85.840,167.954,41.859,157.786
C07854=1031.770,-44.986,-85.852,167.957,41.858,157.786
C07855=1031.775,-44.736,-85.865,167.960,41.857,157.786
C07856=1031.782,-44.487,-85.878,167.962,41.856,157.786
C07857=1031.788,-44.237,-85.890,167.964,41.855,157.786
C07858=1031.794,-43.988,-85.903,167.967,41.853,157.786
C07859=1031.800,-43.738,-85.915,167.970,41.852,157.786
C07860=1031.807,-43.489,-85.928,167.973,41.851,157.786
C07861=1031.813,-43.239,-85.941,167.975,41.850,157.786
C07862=1031.819,-42.989,-85.953,167.978,41.849,157.786
C07863=1031.826,-42.740,-85.966,167.980,41.848,157.785
C07864=1031.832,-42.490,-85.978,167.983,41.847,157.785
C07865=1031.838,-42.240,-85.991,167.986,41.845,157.785
C07866=1031.844,-41.991,-86.004,167.988,41.844,157.785
C07867=1031.851,-41.741,-86.016,167.991,41.843,157.785
C07868=1031.857,-41.492,-86.029,167.994,41.842,157.785
C07869=1031.863,-41.242,-86.042,167.997,41.841,157.785
C07870=1031.869,-40.993,-86.054,167.999,41.840,157.785
C07871=1031.876,-40.743,-86.067,168.001,41.838,157.785
C07872=1031.881,-40.494,-86.080,168.004,41.837,157.785
C07873=1031.887,-40.244,-86.092,168.007,41.836,157.785
C07874=1031.894,-39.995,-86.105,168.010,41.835,157.785
C07875=1031.900,-39.745,-86.117,168.012,41.834,157.785
C07876=1031.906,-39.496,-86.131,168.014,41.833,157.785
C07877=1031.912,-39.246,-86.143,168.017,41.831,157.785
C07878=1031.919,-38.997,-86.156,168.020,41.830,157.785
C07879=1031.926,-38.746,-86.169,168.023,41.829,157.785
C07880=1031.932,-38.497,-86.182,168.025,41.828,157.785
C07881=1031.938,-38.247,-86.195,168.028,41.827,157.785
C07882=1031.944,-37.998,-86.208,168.030,41.826,157.785
C07883=1031.950,-37.748,-86.221,168.032,41.825,157.785
C07884=1031.956,-37.499,-86.234,168.035,41.824,157.785
C07885=1031.962,-37.249,-86.246,168.038,41.823,157.785
C07886=1031.968,-36.999,-86.260,168.041,41.822,157.785
C07887=1031.975,-36.750,-86.273,168.043,41.821,157.784
C07888=1031.982,-36.469,-86.287,168.046,41.820,157.784
C07889=1031.989,-36.188,-86.301,168.049,41.819,157.784
C07890=1031.995,-35.908,-86.317,168.051,41.817,157.784
C07891=1032.002,-35.626,-86.331,168.055,41.816,157.784
C07892=1032.009,-35.377,-86.344,168.057,41.815,157.784
C07893=1032.015,-35.128,-86.358,168.060,41.814,157.784
C07894=1032.021,-34.878,-86.370,168.063,41.813,157.784
C07895=1032.027,-34.629,-86.384,168.065,41.812,157.784
C07896=1032.034,-34.379,-86.397,168.067,41.811,157.784
C07897=1032.040,-34.129,-86.410,168.070,41.809,157.784
C07898=1032.046,-33.879,-86.423,168.073,41.808,157.784
C07899=1032.052,-33.630,-86.436,168.075,41.807,157.784
C07900=1032.058,-33.380,-86.449,168.078,41.806,157.784
C07901=1032.064,-33.131,-86.462,168.081,41.805,157.784
C07902=1032.071,-32.881,-86.476,168.083,41.804,157.784
C07903=1032.077,-32.631,-86.488,168.086,41.803,157.784
C07904=1032.083,-32.382,-86.502,168.088,41.802,157.784
C07905=1032.089,-32.133,-86.515,168.091,41.801,157.784
C07906=1032.096,-31.883,-86.528,168.093,41.800,157.784
C07907=1032.102,-31.633,-86.541,168.096,41.799,157.784
C07908=1032.108,-31.384,-86.554,168.099,41.798,157.784
C07909=1032.115,-31.134,-86.568,168.101,41.797,157.784
C07910=1032.121,-30.885,-86.581,168.104,41.796,157.784
C07911=1032.127,-30.634,-86.594,168.107,41.795,157.784
C07912=1032.133,-30.385,-86.607,168.108,41.794,157.784
C07913=1032.140,-30.136,-86.620,168.111,41.793,157.784
C07914=1032.146,-29.887,-86.634,168.114,41.792,157.784
C07915=1032.153,-29.637,-86.647,168.117,41.791,157.784
C07916=1032.159,-29.387,-86.660,168.119,41.790,157.784
C07917=1032.165,-29.138,-86.673,168.122,41.788,157.783
C07918=1032.171,-28.888,-86.686,168.124,41.787,157.783
C07919=1032.178,-28.638,-86.700,168.126,41.786,157.783
C07920=1032.184,-28.389,-86.713,168.129,41.785,157.783
C07921=1032.190,-28.140,-86.726,168.132,41.784,157.783
C07922=1032.197,-27.890,-86.740,168.135,41.783,157.783
C07923=1032.203,-27.640,-86.753,168.137,41.782,157.783
C07924=1032.209,-27.391,-86.766,168.140,41.781,157.783
C07925=1032.215,-27.141,-86.779,168.142,41.780,157.783
C07926=1032.221,-26.891,-86.793,168.144,41.779,157.783
C07927=1032.228,-26.642,-86.807,168.147,41.778,157.783
C07928=1032.234,-26.393,-86.820,168.150,41.777,157.783
C07929=1032.240,-26.142,-86.834,168.152,41.776,157.783
C07930=1032.246,-25.893,-86.847,168.155,41.775,157.783
C07931=1032.252,-25.644,-86.861,168.157,41.775,157.783
C07932=1032.259,-25.393,-86.875,168.160,41.773,157.783
C07933=1032.265,-25.144,-86.888,168.163,41.772,157.783
C07934=1032.271,-24.895,-86.901,168.164,41.771,157.783
C07935=1032.277,-24.646,-86.915,168.167,41.770,157.783
C07936=1032.283,-24.395,-86.929,168.170,41.769,157.783
C07937=1032.289,-24.146,-86.942,168.172,41.768,157.783
C07938=1032.296,-23.897,-86.956,168.175,41.767,157.783
C07939=1032.302,-23.647,-86.970,168.178,41.766,157.783
C07940=1032.308,-23.398,-86.984,168.180,41.765,157.783
C07941=1032.314,-23.149,-86.997,168.183,41.765,157.783
C07942=1032.321,-22.899,-87.011,168.185,41.764,157.783
C07943=1032.327,-22.649,-87.025,168.187,41.763,157.783
C07944=1032.334,-22.334,-87.042,168.190,41.762,157.783
C07945=1032.343,-22.019,-87.059,168.194,41.760,157.783
C07946=1032.351,-21.704,-87.076,168.197,41.759,157.783
C07947=1032.359,-21.389,-87.093,168.200,41.758,157.783
C07948=1032.364,-21.156,-87.106,168.203,41.757,157.783
C07949=1032.370,-20.923,-87.119,168.204,41.756,157.783
C07950=1032.376,-20.690,-87.132,168.207,41.755,157.783
C07951=1032.382,-20.458,-87.145,168.209,41.754,157.783
C07952=1032.388,-20.225,-87.158,168.212,41.753,157.783
C07953=1032.394,-19.992,-87.171,168.214,41.752,157.783
C07954=1032.400,-19.759,-87.183,168.217,41.751,157.783
C07955=1032.405,-19.526,-87.196,168.219,41.750,157.783
C07956=1032.412,-19.277,-87.209,168.222,41.749,157.783
C07957=1032.418,-19.027,-87.224,168.224,41.748,157.782
C07958=1032.424,-18.778,-87.237,168.226,41.747,157.782
C07959=1032.431,-18.528,-87.251,168.228,41.746,157.782
C07960=1032.436,-18.278,-87.265,168.231,41.745,157.782
C07961=1032.443,-18.029,-87.279,168.234,41.744,157.782
C07962=1032.450,-17.780,-87.293,168.236,41.743,157.782
C07963=1032.455,-17.530,-87.306,168.239,41.742,157.782
C07964=1032.462,-17.280,-87.320,168.242,41.742,157.782
C07965=1032.469,-17.031,-87.334,168.244,41.741,157.782
C07966=1032.475,-16.781,-87.348,168.247,41.740,157.782
C07967=1032.481,-16.532,-87.362,168.248,41.739,157.782
C07968=1032.488,-16.282,-87.376,168.251,41.738,157.782
C07969=1032.494,-16.033,-87.390,168.254,41.737,157.782
C07970=1032.500,-15.783,-87.403,168.256,41.736,157.782
C07971=1032.507,-15.534,-87.417,168.259,41.735,157.782
C07972=1032.513,-15.284,-87.432,168.261,41.734,157.782
C07973=1032.519,-15.035,-87.445,168.264,41.733,157.782
C07974=1032.526,-14.785,-87.460,168.266,41.732,157.782
C07975=1032.531,-14.535,-87.474,168.269,41.732,157.782
C07976=1032.538,-14.286,-87.487,168.271,41.731,157.782
C07977=1032.544,-14.037,-87.502,168.273,41.730,157.782
C07978=1032.550,-13.787,-87.516,168.276,41.729,157.782
C07979=1032.556,-13.538,-87.530,168.278,41.728,157.782
C07980=1032.562,-13.287,-87.544,168.281,41.727,157.782
C07981=1032.569,-13.038,-87.559,168.284,41.726,157.782
C07982=1032.575,-12.788,-87.573,168.286,41.725,157.782
C07983=1032.582,-12.539,-87.587,168.289,41.724,157.782
C07984=1032.587,-12.290,-87.601,168.290,41.723,157.782
C07985=1032.594,-12.040,-87.616,168.293,41.722,157.782
C07986=1032.600,-11.791,-87.629,168.295,41.722,157.782
C07987=1032.606,-11.541,-87.644,168.298,41.721,157.782
C07988=1032.613,-11.292,-87.657,168.300,41.720,157.782
C07989=1032.619,-11.042,-87.672,168.303,41.719,157.782
C07990=1032.625,-10.792,-87.686,168.306,41.718,157.782
C07991=1032.632,-10.543,-87.700,168.308,41.717,157.782
C07992=1032.638,-10.293,-87.715,168.311,41.716,157.782
C07993=1032.644,-10.044,-87.729,168.313,41.715,157.782
C07994=1032.651,-9.795,-87.744,168.315,41.714,157.782
C07995=1032.656,-9.545,-87.757,168.317,41.713,157.782
C07996=1032.663,-9.296,-87.772,168.320,41.712,157.782
C07997=1032.669,-9.045,-87.786,168.322,41.711,157.782
C07998=1032.675,-8.796,-87.801,168.325,41.710,157.782
C07999=1032.682,-8.546,-87.814,168.327,41.710,157.782
C08000=1032.688,-8.297,-87.829,168.330,41.709,157.782
C08001=1032.694,-8.048,-87.844,168.333,41.708,157.782
C08002=1032.701,-7.798,-87.857,168.335,41.707,157.782
C08003=1032.707,-7.549,-87.872,168.337,41.706,157.782
C08004=1032.714,-7.300,-87.886,168.339,41.705,157.782
C08005=1032.720,-7.049,-87.901,168.342,41.704,157.782
C08006=1032.726,-6.800,-87.915,168.344,41.704,157.782
C08007=1032.733,-6.551,-87.929,168.347,41.703,157.782
C08008=1032.738,-6.301,-87.943,168.349,41.702,157.782
C08009=1032.745,-6.052,-87.958,168.352,41.701,157.782
C08010=1032.752,-5.802,-87.973,168.354,41.700,157.781
C08011=1032.757,-5.553,-87.986,168.357,41.699,157.781
C08012=1032.764,-5.303,-88.001,168.359,41.698,157.781
C08013=1032.771,-5.054,-88.016,168.361,41.697,157.781
C08014=1032.777,-4.804,-88.030,168.364,41.696,157.781
C08015=1032.783,-4.555,-88.044,168.366,41.695,157.781
C08016=1032.790,-4.271,-88.060,168.369,41.694,157.781
C08017=1032.798,-3.989,-88.077,168.372,41.693,157.781
C08018=1032.805,-3.705,-88.094,168.375,41.692,157.781
C08019=1032.812,-3.422,-88.110,168.378,41.691,157.781
C08020=1032.818,-3.172,-88.125,168.380,41.690,157.781
C08021=1032.824,-2.923,-88.140,168.383,41.690,157.781
C08022=1032.831,-2.673,-88.155,168.384,41.689,157.781
C08023=1032.837,-2.424,-88.170,168.387,41.688,157.781
C08024=1032.843,-2.175,-88.184,168.389,41.688,157.781
C08025=1032.849,-1.925,-88.199,168.391,41.687,157.781
C08026=1032.855,-1.675,-88.214,168.394,41.686,157.781
C08027=1032.861,-1.426,-88.228,168.396,41.685,157.781
C08028=1032.867,-1.176,-88.243,168.399,41.684,157.781
C08029=1032.874,-0.927,-88.258,168.401,41.683,157.781
C08030=1032.879,-0.678,-88.272,168.404,41.683,157.781
C08031=1032.886,-0.428,-88.287,168.406,41.682,157.781
C08032=1032.892,-0.178,-88.302,168.409,41.681,157.781
C08033=1032.899,0.071,-88.317,168.410,41.680,157.781
C08034=1032.904,0.320,-88.332,168.413,41.680,157.781
C08035=1032.911,0.570,-88.347,168.415,41.679,157.781
C08036=1032.917,0.820,-88.362,168.418,41.678,157.781
C08037=1032.924,1.069,-88.377,168.420,41.677,157.781
C08038=1032.929,1.318,-88.391,168.423,41.676,157.781
C08039=1032.936,1.568,-88.406,168.425,41.675,157.781
C08040=1032.942,1.818,-88.421,168.427,41.675,157.781
C08041=1032.948,2.067,-88.436,168.430,41.674,157.781
C08042=1032.954,2.316,-88.451,168.432,41.673,157.781
C08043=1032.961,2.566,-88.466,168.435,41.672,157.781
C08044=1032.967,2.816,-88.480,168.437,41.672,157.781
C08045=1032.973,3.065,-88.495,168.440,41.671,157.781
C08046=1032.979,3.314,-88.510,168.441,41.670,157.781
C08047=1032.986,3.564,-88.525,168.444,41.669,157.781
C08048=1032.992,3.813,-88.540,168.446,41.669,157.781
C08049=1032.998,4.063,-88.555,168.449,41.667,157.781
C08050=1033.005,4.313,-88.570,168.451,41.667,157.781
C08051=1033.011,4.561,-88.585,168.453,41.666,157.781
C08052=1033.017,4.811,-88.600,168.456,41.665,157.781
C08053=1033.024,5.060,-88.615,168.458,41.664,157.781
C08054=1033.030,5.310,-88.630,168.461,41.663,157.781
C08055=1033.036,5.560,-88.645,168.463,41.663,157.781
C08056=1033.043,5.809,-88.660,168.466,41.662,157.781
C08057=1033.049,6.058,-88.674,168.467,41.661,157.781
C08058=1033.055,6.308,-88.689,168.470,41.660,157.781
C08059=1033.062,6.557,-88.705,168.472,41.660,157.781
C08060=1033.068,6.807,-88.720,168.475,41.659,157.781
C08061=1033.074,7.056,-88.735,168.477,41.658,157.781
C08062=1033.081,7.306,-88.750,168.480,41.657,157.781
C08063=1033.087,7.556,-88.765,168.482,41.656,157.781
C08064=1033.093,7.805,-88.780,168.484,41.655,157.781
C08065=1033.100,8.054,-88.795,168.487,41.654,157.781
C08066=1033.106,8.303,-88.810,168.488,41.653,157.781
C08067=1033.112,8.553,-88.825,168.492,41.653,157.781
C08068=1033.119,8.803,-88.840,168.493,41.652,157.781
C08069=1033.125,9.052,-88.856,168.496,41.651,157.781
C08070=1033.132,9.301,-88.870,168.498,41.650,157.781
C08071=1033.138,9.551,-88.885,168.501,41.649,157.781
C08072=1033.144,9.801,-88.901,168.503,41.649,157.781
C08073=1033.150,10.051,-88.916,168.505,41.648,157.781
C08074=1033.157,10.300,-88.932,168.508,41.647,157.781
C08075=1033.163,10.549,-88.947,168.510,41.646,157.781
C08076=1033.169,10.798,-88.961,168.513,41.645,157.781
C08077=1033.176,11.047,-88.977,168.515,41.645,157.781
C08078=1033.182,11.297,-88.992,168.517,41.644,157.781
C08079=1033.189,11.547,-89.007,168.519,41.643,157.781
C08080=1033.196,11.832,-89.024,168.522,41.642,157.781
C08081=1033.204,12.117,-89.042,168.525,41.640,157.781
C08082=1033.210,12.402,-89.059,168.528,41.639,157.781
C08083=1033.218,12.687,-89.076,168.530,41.638,157.781
C08084=1033.224,12.936,-89.092,168.533,41.638,157.781
C08085=1033.231,13.186,-89.107,168.535,41.637,157.781
C08086=1033.237,13.436,-89.122,168.537,41.636,157.781
C08087=1033.244,13.685,-89.137,168.539,41.635,157.781
C08088=1033.250,13.934,-89.152,168.542,41.634,157.781
C08089=1033.257,14.184,-89.167,168.544,41.634,157.781
C08090=1033.263,14.433,-89.184,168.546,41.633,157.781
C08091=1033.269,14.683,-89.199,168.549,41.632,157.781
C08092=1033.276,14.932,-89.214,168.551,41.632,157.781
C08093=1033.281,15.182,-89.230,168.554,41.631,157.781
C08094=1033.288,15.431,-89.245,168.556,41.630,157.781
C08095=1033.294,15.681,-89.260,168.558,41.629,157.781
C08096=1033.300,15.930,-89.277,168.561,41.628,157.781
C08097=1033.307,16.180,-89.292,168.563,41.628,157.781
C08098=1033.313,16.429,-89.307,168.566,41.627,157.781
C08099=1033.319,16.679,-89.323,168.567,41.626,157.781
C08100=1033.326,16.928,-89.338,168.569,41.625,157.781
C08101=1033.332,17.177,-89.353,168.572,41.625,157.781
C08102=1033.338,17.427,-89.370,168.574,41.624,157.781
C08103=1033.344,17.677,-89.385,168.577,41.623,157.781
C08104=1033.351,17.926,-89.400,168.579,41.623,157.781
C08105=1033.357,18.175,-89.417,168.581,41.622,157.781
C08106=1033.364,18.425,-89.431,168.584,41.621,157.781
C08107=1033.370,18.674,-89.447,168.586,41.620,157.781
C08108=1033.376,18.924,-89.463,168.588,41.619,157.781
C08109=1033.383,19.173,-89.478,168.591,41.618,157.781
C08110=1033.389,19.422,-89.493,168.593,41.618,157.781
C08111=1033.395,19.672,-89.510,168.595,41.617,157.781
C08112=1033.402,19.921,-89.526,168.597,41.616,157.781
C08113=1033.408,20.171,-89.541,168.599,41.616,157.781
C08114=1033.414,20.420,-89.557,168.602,41.615,157.781
C08115=1033.420,20.670,-89.573,168.604,41.614,157.780
C08116=1033.427,20.919,-89.588,168.606,41.614,157.781
C08117=1033.434,21.168,-89.604,168.609,41.613,157.781
C08118=1033.439,21.418,-89.620,168.611,41.612,157.781
C08119=1033.446,21.667,-89.635,168.614,41.611,157.781
C08120=1033.452,21.917,-89.651,168.616,41.610,157.781
C08121=1033.458,22.166,-89.667,168.618,41.610,157.781
C08122=1033.464,22.415,-89.683,168.621,41.609,157.781
C08123=1033.471,22.665,-89.698,168.622,41.608,157.780
C08124=1033.477,22.914,-89.714,168.624,41.608,157.781
C08125=1033.484,23.164,-89.730,168.627,41.607,157.781
C08126=1033.490,23.413,-89.747,168.629,41.606,157.780
C08127=1033.496,23.663,-89.761,168.631,41.606,157.781
C08128=1033.502,23.912,-89.778,168.634,41.604,157.781
C08129=1033.509,24.161,-89.793,168.636,41.604,157.780
C08130=1033.515,24.411,-89.810,168.639,41.603,157.781
C08131=1033.521,24.660,-89.825,168.641,41.602,157.780
C08132=1033.527,24.910,-89.841,168.643,41.601,157.780
C08133=1033.535,25.159,-89.857,168.646,41.601,157.781
C08134=1033.541,25.409,-89.873,168.648,41.600,157.780
C08135=1033.547,25.658,-89.889,168.649,41.599,157.780
C08136=1033.553,25.908,-89.904,168.653,41.599,157.781
C08137=1033.560,26.157,-89.920,168.654,41.598,157.780
C08138=1033.566,26.406,-89.936,168.656,41.597,157.780
C08139=1033.573,26.656,-89.952,168.659,41.596,157.781
C08140=1033.579,26.905,-89.969,168.661,41.596,157.780
C08141=1033.585,27.155,-89.985,168.664,41.595,157.781
C08142=1033.591,27.404,-90.000,168.666,41.594,157.780
C08143=1033.597,27.653,-90.017,168.668,41.593,157.780
C08144=1033.604,27.940,-90.035,168.671,41.592,157.780
C08145=1033.612,28.226,-90.053,168.674,41.592,157.780
C08146=1033.619,28.512,-90.072,168.676,41.591,157.780
C08147=1033.626,28.799,-90.090,168.679,41.590,157.780
C08148=1033.632,29.048,-90.106,168.681,41.590,157.780
C08149=1033.639,29.298,-90.122,168.683,41.589,157.780
C08150=1033.646,29.548,-90.138,168.685,41.588,157.781
C08151=1033.651,29.797,-90.155,168.687,41.587,157.780
C08152=1033.657,30.046,-90.171,168.690,41.587,157.781
C08153=1033.664,30.295,-90.187,168.692,41.586,157.780
C08154=1033.670,30.545,-90.203,168.694,41.585,157.780
C08155=1033.676,30.794,-90.219,168.697,41.585,157.781
C08156=1033.683,31.044,-90.235,168.699,41.584,157.780
C08157=1033.689,31.293,-90.251,168.701,41.584,157.781
C08158=1033.696,31.542,-90.268,168.703,41.583,157.780
C08159=1033.701,31.791,-90.285,168.706,41.582,157.781
C08160=1033.709,32.041,-90.301,168.708,41.581,157.781
C08161=1033.715,32.290,-90.317,168.710,41.580,157.780
C08162=1033.721,32.540,-90.333,168.713,41.580,157.781
C08163=1033.727,32.789,-90.349,168.714,41.579,157.781
C08164=1033.734,33.039,-90.365,168.717,41.579,157.781
C08165=1033.740,33.288,-90.382,168.719,41.578,157.781
C08166=1033.746,33.537,-90.398,168.721,41.577,157.780
C08167=1033.752,33.787,-90.414,168.723,41.577,157.781
C08168=1033.759,34.036,-90.430,168.726,41.576,157.781
C08169=1033.765,34.285,-90.447,168.728,41.575,157.781
C08170=1033.771,34.535,-90.463,168.730,41.574,157.781
C08171=1033.777,34.784,-90.480,168.733,41.573,157.781
C08172=1033.785,35.034,-90.496,168.735,41.573,157.781
C08173=1033.790,35.283,-90.512,168.737,41.572,157.781
C08174=1033.796,35.532,-90.528,168.740,41.571,157.780
C08175=1033.803,35.782,-90.545,168.742,41.571,157.781
C08176=1033.810,36.031,-90.561,168.744,41.570,157.780
C08177=1033.816,36.280,-90.577,168.747,41.570,157.781
C08178=1033.822,36.530,-90.594,168.748,41.569,157.781
C08179=1033.828,36.780,-90.610,168.750,41.568,157.780
C08180=1033.834,37.029,-90.627,168.753,41.567,157.781
C08181=1033.842,37.278,-90.643,168.755,41.566,157.781
C08182=1033.848,37.527,-90.660,168.757,41.565,157.780
C08183=1033.854,37.777,-90.676,168.759,41.565,157.781
C08184=1033.860,38.026,-90.692,168.762,41.564,157.780
C08185=1033.867,38.275,-90.709,168.764,41.564,157.781
C08186=1033.873,38.525,-90.726,168.766,41.563,157.780
C08187=1033.879,38.774,-90.742,168.769,41.563,157.781
C08188=1033.885,39.024,-90.759,168.771,41.562,157.781
C08189=1033.891,39.273,-90.776,168.773,41.561,157.781
C08190=1033.897,39.522,-90.792,168.775,41.561,157.781
C08191=1033.904,39.772,-90.809,168.778,41.560,157.781
C08192=1033.910,40.021,-90.825,168.780,41.559,157.781
C08193=1033.916,40.270,-90.842,168.782,41.559,157.781
C08194=1033.923,40.520,-90.859,168.784,41.558,157.781
C08195=1033.929,40.769,-90.875,168.786,41.558,157.781
C08196=1033.935,41.019,-90.892,168.788,41.557,157.781
C08197=1033.942,41.268,-90.909,168.790,41.556,157.781
C08198=1033.948,41.517,-90.925,168.793,41.555,157.781
C08199=1033.955,41.767,-90.942,168.795,41.554,157.781
C08200=1033.960,42.016,-90.959,168.797,41.554,157.781
C08201=1033.966,42.265,-90.975,168.800,41.553,157.781
C08202=1033.973,42.515,-90.992,168.802,41.553,157.781
C08203=1033.979,42.764,-91.009,168.804,41.552,157.781
C08204=1033.985,43.013,-91.026,168.806,41.552,157.781
C08205=1033.992,43.263,-91.042,168.809,41.551,157.781
C08206=1033.998,43.512,-91.060,168.811,41.550,157.781
C08207=1034.004,43.762,-91.076,168.813,41.550,157.781
C08208=1034.011,44.048,-91.096,168.816,41.549,157.781
C08209=1034.018,44.335,-91.116,168.818,41.549,157.781
C08210=1034.025,44.621,-91.134,168.821,41.548,157.781
C08211=1034.032,44.907,-91.154,168.823,41.548,157.781
C08212=1034.039,45.157,-91.171,168.825,41.546,157.781
C08213=1034.044,45.406,-91.188,168.827,41.546,157.781
C08214=1034.050,45.655,-91.205,168.829,41.545,157.781
C08215=1034.057,45.905,-91.222,168.831,41.545,157.781
C08216=1034.063,46.153,-91.239,168.834,41.544,157.781
C08217=1034.069,46.404,-91.256,168.836,41.544,157.781
C08218=1034.075,46.652,-91.273,168.838,41.543,157.781
C08219=1034.082,46.901,-91.290,168.840,41.543,157.781
C08220=1034.088,47.151,-91.307,168.843,41.542,157.781
C08221=1034.094,47.400,-91.324,168.845,41.541,157.781
C08222=1034.100,47.650,-91.341,168.847,41.541,157.781
C08223=1034.106,47.899,-91.358,168.849,41.540,157.781
C08224=1034.113,48.149,-91.376,168.852,41.540,157.781
C08225=1034.119,48.398,-91.392,168.854,41.539,157.781
C08226=1034.125,48.647,-91.409,168.856,41.539,157.781
C08227=1034.132,48.896,-91.426,168.858,41.538,157.781
C08228=1034.137,49.146,-91.443,168.861,41.537,157.781
C08229=1034.144,49.395,-91.461,168.863,41.537,157.781
C08230=1034.150,49.644,-91.477,168.865,41.536,157.781
C08231=1034.156,49.894,-91.495,168.867,41.536,157.781
C08232=1034.162,50.143,-91.512,168.870,41.535,157.781
C08233=1034.169,50.393,-91.529,168.872,41.534,157.781
C08234=1034.175,50.641,-91.546,168.873,41.534,157.781
C08235=1034.181,50.892,-91.563,168.875,41.533,157.781
C08236=1034.187,51.140,-91.580,168.878,41.532,157.781
C08237=1034.194,51.390,-91.598,168.880,41.532,157.781
C08238=1034.200,51.639,-91.615,168.882,41.531,157.781
C08239=1034.206,51.889,-91.632,168.884,41.531,157.781
C08240=1034.212,52.138,-91.649,168.887,41.530,157.781
C08241=1034.219,52.387,-91.667,168.889,41.530,157.781
C08242=1034.225,52.636,-91.684,168.891,41.529,157.781
C08243=1034.231,52.886,-91.700,168.893,41.528,157.781
C08244=1034.237,53.135,-91.718,168.896,41.527,157.781
C08245=1034.244,53.385,-91.735,168.898,41.527,157.781
C08246=1034.250,53.633,-91.752,168.900,41.526,157.781
C08247=1034.257,53.883,-91.769,168.902,41.526,157.781
C08248=1034.262,54.133,-91.786,168.905,41.525,157.781
C08249=1034.269,54.382,-91.804,168.907,41.525,157.781
C08250=1034.276,54.631,-91.821,168.909,41.524,157.781
C08251=1034.281,54.880,-91.839,168.911,41.523,157.781
C08252=1034.288,55.130,-91.856,168.913,41.522,157.781
C08253=1034.294,55.379,-91.873,168.915,41.522,157.781
C08254=1034.301,55.628,-91.891,168.917,41.521,157.781
C08255=1034.306,55.878,-91.907,168.919,41.521,157.781
C08256=1034.313,56.127,-91.924,168.922,41.520,157.781
C08257=1034.319,56.377,-91.942,168.924,41.520,157.782
C08258=1034.326,56.626,-91.959,168.926,41.519,157.781
C08259=1034.333,56.875,-91.977,168.929,41.518,157.782
C08260=1034.338,57.124,-91.994,168.931,41.517,157.781
C08261=1034.345,57.373,-92.012,168.933,41.516,157.781
C08262=1034.352,57.623,-92.029,168.935,41.516,157.781
C08263=1034.357,57.872,-92.046,168.938,41.515,157.781
C08264=1034.364,58.121,-92.064,168.940,41.515,157.782
C08265=1034.370,58.371,-92.080,168.942,41.514,157.781
C08266=1034.376,58.620,-92.098,168.944,41.514,157.782
C08267=1034.383,58.870,-92.115,168.947,41.513,157.781
C08268=1034.389,59.119,-92.132,168.949,41.512,157.782
C08269=1034.395,59.368,-92.150,168.950,41.511,157.781
C08270=1034.402,59.618,-92.168,168.952,41.511,157.781
C08271=1034.409,59.867,-92.184,168.955,41.510,157.782
C08272=1034.416,60.153,-92.205,168.957,41.509,157.781
C08273=1034.423,60.439,-92.225,168.960,41.509,157.782
C08274=1034.430,60.725,-92.245,168.963,41.508,157.782
C08275=1034.439,61.011,-92.265,168.965,41.507,157.781
C08276=1034.444,61.260,-92.283,168.967,41.507,157.782
C08277=1034.451,61.509,-92.300,168.970,41.506,157.781
C08278=1034.457,61.759,-92.318,168.972,41.505,157.781
C08279=1034.463,62.008,-92.335,168.974,41.504,157.781
C08280=1034.470,62.257,-92.352,168.977,41.503,157.781
C08281=1034.476,62.507,-92.370,168.979,41.503,157.782
C08282=1034.483,62.756,-92.388,168.980,41.502,157.781
C08283=1034.490,63.005,-92.405,168.982,41.501,157.781
C08284=1034.496,63.255,-92.422,168.985,41.501,157.781
C08285=1034.503,63.504,-92.440,168.987,41.500,157.781
C08286=1034.508,63.753,-92.457,168.989,41.500,157.781
C08287=1034.515,64.003,-92.475,168.991,41.499,157.781
C08288=1034.521,64.252,-92.493,168.994,41.498,157.782
C08289=1034.528,64.501,-92.511,168.996,41.498,157.781
C08290=1034.534,64.750,-92.528,168.998,41.497,157.782
C08291=1034.540,65.000,-92.546,169.000,41.497,157.782
C08292=1034.547,65.249,-92.564,169.003,41.496,157.782
C08293=1034.552,65.498,-92.581,169.005,41.496,157.782
C08294=1034.559,65.748,-92.600,169.007,41.495,157.782
C08295=1034.565,65.997,-92.617,169.009,41.495,157.782
C08296=1034.571,66.246,-92.635,169.012,41.494,157.782
C08297=1034.578,66.495,-92.652,169.014,41.493,157.782
C08298=1034.584,66.745,-92.671,169.016,41.492,157.782
C08299=1034.590,66.994,-92.689,169.018,41.492,157.782
C08300=1034.596,67.243,-92.706,169.019,41.491,157.782
C08301=1034.603,67.493,-92.723,169.023,41.491,157.782
C08302=1034.609,67.742,-92.742,169.025,41.491,157.782
C08303=1034.615,67.992,-92.760,169.026,41.490,157.782
C08304=1034.622,68.240,-92.777,169.028,41.489,157.782
C08305=1034.628,68.490,-92.796,169.031,41.488,157.782
C08306=1034.634,68.739,-92.814,169.033,41.488,157.782
C08307=1034.641,68.989,-92.831,169.035,41.487,157.782
C08308=1034.647,69.237,-92.849,169.037,41.487,157.782
C08309=1034.653,69.487,-92.867,169.040,41.486,157.782
C08310=1034.659,69.737,-92.885,169.042,41.486,157.782
C08311=1034.665,69.986,-92.904,169.044,41.485,157.782
C08312=1034.672,70.234,-92.921,169.046,41.484,157.782
C08313=1034.678,70.484,-92.939,169.048,41.484,157.782
C08314=1034.684,70.733,-92.957,169.051,41.483,157.782
C08315=1034.690,70.983,-92.975,169.053,41.483,157.782
C08316=1034.696,71.231,-92.994,169.055,41.483,157.782
C08317=1034.702,71.481,-93.011,169.057,41.482,157.782
C08318=1034.710,71.730,-93.030,169.060,41.481,157.782
C08319=1034.716,71.980,-93.047,169.062,41.480,157.782
C08320=1034.722,72.229,-93.066,169.064,41.480,157.782
C08321=1034.728,72.478,-93.084,169.066,41.480,157.782
C08322=1034.734,72.728,-93.102,169.068,41.479,157.782
C08323=1034.740,72.977,-93.120,169.071,41.479,157.782
C08324=1034.746,73.227,-93.138,169.072,41.478,157.782
C08325=1034.753,73.476,-93.157,169.075,41.477,157.782
C08326=1034.759,73.724,-93.174,169.077,41.477,157.782
C08327=1034.765,73.974,-93.192,169.079,41.476,157.782
C08328=1034.771,74.223,-93.210,169.081,41.476,157.782
C08329=1034.778,74.472,-93.229,169.083,41.475,157.782
C08330=1034.784,74.722,-93.247,169.085,41.475,157.782
C08331=1034.790,74.971,-93.266,169.087,41.474,157.782
C08332=1034.796,75.220,-93.284,169.090,41.473,157.782
C08333=1034.802,75.469,-93.302,169.092,41.473,157.782
C08334=1034.810,75.718,-93.320,169.094,41.472,157.782
C08335=1034.816,75.968,-93.338,169.096,41.472,157.782
C08336=1034.822,76.254,-93.359,169.099,41.471,157.782
C08337=1034.830,76.540,-93.380,169.101,41.471,157.782
C08338=1034.837,76.825,-93.401,169.104,41.470,157.782
C08339=1034.844,77.111,-93.422,169.107,41.469,157.782
C08340=1034.851,77.361,-93.440,169.109,41.468,157.782
C08341=1034.856,77.609,-93.459,169.111,41.468,157.782
C08342=1034.863,77.859,-93.477,169.113,41.468,157.782
C08343=1034.869,78.108,-93.495,169.115,41.467,157.782
C08344=1034.875,78.357,-93.514,169.118,41.466,157.783
C08345=1034.882,78.607,-93.532,169.120,41.466,157.783
C08346=1034.888,78.856,-93.550,169.122,41.465,157.783
C08347=1034.894,79.105,-93.569,169.124,41.465,157.783
C08348=1034.900,79.355,-93.588,169.126,41.465,157.783
C08349=1034.906,79.604,-93.606,169.129,41.464,157.783
C08350=1034.912,79.853,-93.625,169.131,41.464,157.783
C08351=1034.918,80.102,-93.643,169.133,41.463,157.783
C08352=1034.925,80.351,-93.662,169.134,41.462,157.783
C08353=1034.931,80.601,-93.680,169.136,41.462,157.783
C08354=1034.937,80.850,-93.698,169.139,41.462,157.783
C08355=1034.943,81.099,-93.718,169.142,41.461,157.783
C08356=1034.950,81.349,-93.736,169.143,41.461,157.783
C08357=1034.956,81.598,-93.754,169.145,41.460,157.783
C08358=1034.961,81.847,-93.773,169.148,41.460,157.783
C08359=1034.968,82.096,-93.791,169.150,41.459,157.783
C08360=1034.974,82.345,-93.810,169.152,41.459,157.783
C08361=1034.980,82.594,-93.829,169.154,41.458,157.783
C08362=1034.986,82.844,-93.848,169.156,41.458,157.783
C08363=1034.993,83.093,-93.866,169.159,41.457,157.783
C08364=1034.999,83.342,-93.884,169.161,41.456,157.783
C08365=1035.005,83.592,-93.903,169.163,41.456,157.783
C08366=1035.012,83.841,-93.922,169.165,41.456,157.783
C08367=1035.018,84.090,-93.940,169.167,41.455,157.783
C08368=1035.024,84.339,-93.959,169.170,41.454,157.783
C08369=1035.030,84.588,-93.978,169.172,41.454,157.783
C08370=1035.036,84.838,-93.996,169.174,41.453,157.783
C08371=1035.043,85.087,-94.015,169.176,41.453,157.783
C08372=1035.049,85.336,-94.033,169.179,41.453,157.783
C08373=1035.055,85.586,-94.053,169.181,41.452,157.783
C08374=1035.061,85.835,-94.071,169.183,41.451,157.783
C08375=1035.068,86.084,-94.090,169.185,41.451,157.783
C08376=1035.074,86.333,-94.109,169.188,41.450,157.783
C08377=1035.081,86.582,-94.127,169.190,41.450,157.783
C08378=1035.087,86.831,-94.146,169.192,41.449,157.783
C08379=1035.093,87.081,-94.165,169.194,41.449,157.783
C08380=1035.099,87.330,-94.184,169.196,41.448,157.784
C08381=1035.106,87.579,-94.202,169.199,41.447,157.783
C08382=1035.112,87.828,-94.221,169.201,41.447,157.784
C08383=1035.119,88.077,-94.240,169.202,41.446,157.783
C08384=1035.124,88.327,-94.259,169.204,41.446,157.784
C08385=1035.130,88.576,-94.277,169.208,41.446,157.784
C08386=1035.137,88.826,-94.296,169.209,41.445,157.784
C08387=1035.143,89.075,-94.314,169.211,41.444,157.784
C08388=1035.150,89.323,-94.334,169.213,41.444,157.784
C08389=1035.156,89.573,-94.353,169.216,41.443,157.784
C08390=1035.162,89.822,-94.371,169.218,41.443,157.784
C08391=1035.168,90.071,-94.390,169.220,41.442,157.784
C08392=1035.174,90.320,-94.409,169.222,41.442,157.784
C08393=1035.181,90.569,-94.428,169.225,41.441,157.784
C08394=1035.187,90.819,-94.447,169.227,41.440,157.784
C08395=1035.193,91.068,-94.466,169.229,41.440,157.784
C08396=1035.199,91.317,-94.485,169.231,41.440,157.784
C08397=1035.205,91.567,-94.504,169.233,41.440,157.784
C08398=1035.212,91.815,-94.523,169.236,41.439,157.784
C08399=1035.217,92.064,-94.542,169.238,41.438,157.784
C08400=1035.224,92.351,-94.564,169.240,41.438,157.784
C08401=1035.232,92.637,-94.586,169.243,41.438,157.784
C08402=1035.238,92.922,-94.608,169.245,41.437,157.784
C08403=1035.246,93.208,-94.630,169.248,41.436,157.784
C08404=1035.252,93.457,-94.649,169.250,41.436,157.784
C08405=1035.258,93.706,-94.668,169.252,41.435,157.784
C08406=1035.264,93.956,-94.686,169.255,41.435,157.784
C08407=1035.270,94.204,-94.706,169.257,41.435,157.784
C08408=1035.277,94.453,-94.725,169.259,41.434,157.784
C08409=1035.282,94.703,-94.744,169.261,41.433,157.784
C08410=1035.289,94.953,-94.763,169.263,41.433,157.784
C08411=1035.295,95.202,-94.783,169.266,41.433,157.784
C08412=1035.302,95.451,-94.802,169.268,41.432,157.784
C08413=1035.308,95.700,-94.821,169.270,41.432,157.784
C08414=1035.314,95.949,-94.840,169.272,41.431,157.785
C08415=1035.320,96.198,-94.860,169.275,41.430,157.785
C08416=1035.326,96.447,-94.878,169.277,41.430,157.785
C08417=1035.332,96.697,-94.898,169.279,41.430,157.785
C08418=1035.339,96.946,-94.917,169.281,41.430,157.785
C08419=1035.345,97.195,-94.937,169.284,41.429,157.785
C08420=1035.352,97.444,-94.955,169.286,41.428,157.785
C08421=1035.358,97.693,-94.975,169.288,41.428,157.785
C08422=1035.364,97.942,-94.994,169.290,41.427,157.785
C08423=1035.370,98.192,-95.013,169.293,41.427,157.785
C08424=1035.376,98.440,-95.033,169.295,41.427,157.785
C08425=1035.383,98.690,-95.052,169.296,41.426,157.785
C08426=1035.389,98.939,-95.071,169.298,41.425,157.785
C08427=1035.395,99.188,-95.091,169.302,41.425,157.785
C08428=1035.402,99.437,-95.109,169.303,41.424,157.785
C08429=1035.407,99.687,-95.129,169.305,41.424,157.785
C08430=1035.414,99.935,-95.148,169.307,41.424,157.785
C08431=1035.420,100.185,-95.168,169.310,41.422,157.785
C08432=1035.426,100.434,-95.188,169.312,41.422,157.785
C08433=1035.433,100.683,-95.206,169.314,41.422,157.785
C08434=1035.439,100.932,-95.226,169.316,41.422,157.785
C08435=1035.444,101.182,-95.245,169.318,41.421,157.785
C08436=1035.450,101.430,-95.265,169.321,41.421,157.785
C08437=1035.457,101.680,-95.284,169.323,41.420,157.785
C08438=1035.463,101.929,-95.304,169.325,41.420,157.785
C08439=1035.469,102.179,-95.324,169.327,41.420,157.785
C08440=1035.475,102.427,-95.344,169.330,41.419,157.786
C08441=1035.481,102.677,-95.363,169.332,41.419,157.786
C08442=1035.488,102.926,-95.383,169.334,41.418,157.786
C08443=1035.494,103.175,-95.402,169.336,41.418,157.786
C08444=1035.500,103.424,-95.422,169.338,41.418,157.786
C08445=1035.506,103.673,-95.442,169.341,41.417,157.786
C08446=1035.512,103.922,-95.460,169.343,41.417,157.786
C08447=1035.519,104.172,-95.481,169.345,41.416,157.786
C08448=1035.524,104.421,-95.500,169.347,41.416,157.786
C08449=1035.530,104.670,-95.520,169.350,41.415,157.786
C08450=1035.536,104.919,-95.539,169.352,41.415,157.786
C08451=1035.543,105.168,-95.558,169.354,41.414,157.786
C08452=1035.549,105.417,-95.579,169.356,41.414,157.786
C08453=1035.555,105.667,-95.598,169.359,41.414,157.786
C08454=1035.561,105.916,-95.618,169.361,41.413,157.786
C08455=1035.567,106.164,-95.638,169.363,41.413,157.786
C08456=1035.574,106.414,-95.657,169.365,41.412,157.786
C08457=1035.580,106.663,-95.677,169.368,41.412,157.786
C08458=1035.586,106.912,-95.697,169.370,41.412,157.786
C08459=1035.592,107.161,-95.716,169.372,41.411,157.786
C08460=1035.599,107.410,-95.736,169.374,41.410,157.786
C08461=1035.605,107.659,-95.756,169.377,41.410,157.786
C08462=1035.611,107.909,-95.775,169.379,41.410,157.786
C08463=1035.617,108.158,-95.795,169.381,41.409,157.786
C08464=1035.625,108.444,-95.818,169.384,41.408,157.786
C08465=1035.632,108.730,-95.841,169.386,41.408,157.787
C08466=1035.639,109.016,-95.863,169.389,41.408,157.787
C08467=1035.646,109.302,-95.886,169.392,41.407,157.787
C08468=1035.652,109.550,-95.905,169.394,41.407,157.787
C08469=1035.658,109.799,-95.925,169.396,41.406,157.787
C08470=1035.665,110.049,-95.946,169.398,41.406,157.787
C08471=1035.671,110.298,-95.965,169.401,41.406,157.787
C08472=1035.677,110.547,-95.985,169.403,41.405,157.787
C08473=1035.683,110.796,-96.005,169.405,41.404,157.787
C08474=1035.689,111.045,-96.025,169.407,41.404,157.787
C08475=1035.695,111.294,-96.045,169.410,41.404,157.787
C08476=1035.702,111.544,-96.065,169.412,41.404,157.787
C08477=1035.708,111.793,-96.085,169.414,41.403,157.787
C08478=1035.714,112.042,-96.105,169.416,41.402,157.787
C08479=1035.720,112.291,-96.125,169.419,41.402,157.787
C08480=1035.726,112.540,-96.145,169.421,41.402,157.787
C08481=1035.732,112.789,-96.165,169.423,41.401,157.787
C08482=1035.739,113.038,-96.185,169.426,41.401,157.787
C08483=1035.745,113.287,-96.205,169.428,41.400,157.787
C08484=1035.751,113.536,-96.225,169.430,41.400,157.787
C08485=1035.757,113.785,-96.245,169.432,41.400,157.787
C08486=1035.763,114.034,-96.265,169.434,41.399,157.788
C08487=1035.769,114.283,-96.285,169.437,41.399,157.788
C08488=1035.775,114.533,-96.306,169.439,41.399,157.788
C08489=1035.781,114.782,-96.326,169.441,41.399,157.788
C08490=1035.787,115.031,-96.346,169.443,41.398,157.788
C08491=1035.794,115.280,-96.366,169.446,41.398,157.788
C08492=1035.799,115.529,-96.387,169.448,41.398,157.788
C08493=1035.805,115.778,-96.407,169.450,41.397,157.788
C08494=1035.812,116.028,-96.427,169.452,41.397,157.788
C08495=1035.818,116.276,-96.447,169.455,41.397,157.788
C08496=1035.823,116.525,-96.468,169.457,41.396,157.788
C08497=1035.829,116.775,-96.488,169.459,41.396,157.788
C08498=1035.835,117.024,-96.508,169.461,41.396,157.788
C08499=1035.841,117.273,-96.528,169.464,41.396,157.788
C08500=1035.847,117.522,-96.549,169.466,41.395,157.789
C08501=1035.853,117.771,-96.569,169.468,41.395,157.789
C08502=1035.860,118.021,-96.589,169.470,41.394,157.789
C08503=1035.866,118.269,-96.610,169.473,41.394,157.789
C08504=1035.871,118.518,-96.631,169.475,41.394,157.789
C08505=1035.878,118.768,-96.651,169.477,41.393,157.789
C08506=1035.884,119.016,-96.671,169.479,41.393,157.789
C08507=1035.890,119.266,-96.692,169.482,41.393,157.789
C08508=1035.896,119.515,-96.712,169.484,41.392,157.789
C08509=1035.902,119.764,-96.732,169.486,41.392,157.789
C08510=1035.909,120.013,-96.753,169.490,41.392,157.789
C08511=1035.914,120.262,-96.773,169.492,41.391,157.789
C08512=1035.921,120.511,-96.794,169.494,41.391,157.789
C08513=1035.927,120.760,-96.814,169.496,41.391,157.789
C08514=1035.933,121.010,-96.834,169.499,41.391,157.789
C08515=1035.939,121.258,-96.855,169.500,41.390,157.789
C08516=1035.945,121.507,-96.875,169.503,41.389,157.789
C08517=1035.951,121.757,-96.895,169.506,41.389,157.789
C08518=1035.957,122.006,-96.916,169.508,41.389,157.790
C08519=1035.963,122.255,-96.936,169.510,41.389,157.790
C08520=1035.970,122.503,-96.957,169.512,41.388,157.790
C08521=1035.976,122.753,-96.977,169.515,41.388,157.790
C08522=1035.981,123.002,-96.998,169.517,41.388,157.790
C08523=1035.988,123.251,-97.019,169.519,41.387,157.790
C08524=1035.994,123.500,-97.039,169.522,41.387,157.790
C08525=1036.000,123.750,-97.060,169.524,41.387,157.790
C08526=1036.006,123.998,-97.080,169.526,41.386,157.790
C08527=1036.013,124.247,-97.101,169.529,41.385,157.790
C08528=1036.020,124.533,-97.124,169.531,41.385,157.790
C08529=1036.027,124.819,-97.147,169.534,41.385,157.790
C08530=1036.034,125.104,-97.171,169.537,41.384,157.790
C08531=1036.041,125.390,-97.195,169.539,41.384,157.790
C08532=1036.047,125.639,-97.215,169.542,41.384,157.790
C08533=1036.053,125.888,-97.237,169.544,41.383,157.791
C08534=1036.059,126.137,-97.257,169.546,41.383,157.791
C08535=1036.066,126.386,-97.277,169.548,41.382,157.791
C08536=1036.072,126.635,-97.298,169.551,41.382,157.791
C08537=1036.078,126.885,-97.318,169.553,41.382,157.791
C08538=1036.085,127.133,-97.340,169.555,41.381,157.791
C08539=1036.091,127.382,-97.359,169.558,41.381,157.791
C08540=1036.097,127.632,-97.380,169.560,41.381,157.791
C08541=1036.103,127.880,-97.401,169.563,41.380,157.791
C08542=1036.110,128.130,-97.421,169.565,41.380,157.791
C08543=1036.115,128.378,-97.443,169.567,41.380,157.791
C08544=1036.122,128.628,-97.463,169.570,41.379,157.791
C08545=1036.129,128.877,-97.483,169.572,41.379,157.791
C08546=1036.134,129.126,-97.505,169.574,41.378,157.791
C08547=1036.141,129.375,-97.525,169.577,41.378,157.791
C08548=1036.148,129.624,-97.546,169.579,41.378,157.791
C08549=1036.153,129.873,-97.567,169.581,41.377,157.791
C08550=1036.160,130.122,-97.588,169.584,41.377,157.792
C08551=1036.166,130.371,-97.608,169.586,41.377,157.792
C08552=1036.173,130.620,-97.629,169.588,41.376,157.792
C08553=1036.179,130.870,-97.649,169.591,41.376,157.792
C08554=1036.185,131.118,-97.670,169.593,41.375,157.792
C08555=1036.191,131.368,-97.691,169.595,41.375,157.792
C08556=1036.197,131.617,-97.713,169.598,41.375,157.792
C08557=1036.203,131.865,-97.733,169.600,41.375,157.792
C08558=1036.209,132.115,-97.754,169.602,41.375,157.792
C08559=1036.215,132.363,-97.776,169.605,41.374,157.792
C08560=1036.222,132.612,-97.797,169.607,41.374,157.792
C08561=1036.227,132.862,-97.818,169.609,41.374,157.792
C08562=1036.233,133.111,-97.839,169.612,41.373,157.792
C08563=1036.240,133.360,-97.860,169.614,41.373,157.792
C08564=1036.245,133.609,-97.880,169.616,41.373,157.793
C08565=1036.252,133.858,-97.901,169.619,41.373,157.793
C08566=1036.258,134.107,-97.923,169.621,41.372,157.793
C08567=1036.263,134.356,-97.944,169.623,41.372,157.793
C08568=1036.270,134.605,-97.965,169.626,41.372,157.793
C08569=1036.276,134.854,-97.986,169.629,41.371,157.793
C08570=1036.282,135.103,-98.007,169.631,41.371,157.793
C08571=1036.289,135.352,-98.028,169.634,41.371,157.793
C08572=1036.295,135.601,-98.050,169.636,41.371,157.793
C08573=1036.300,135.850,-98.071,169.639,41.370,157.793
C08574=1036.307,136.099,-98.091,169.641,41.370,157.793
C08575=1036.313,136.349,-98.113,169.643,41.370,157.793
C08576=1036.319,136.597,-98.134,169.646,41.369,157.793
C08577=1036.326,136.846,-98.155,169.648,41.369,157.794
C08578=1036.332,137.095,-98.177,169.650,41.369,157.794
C08579=1036.338,137.345,-98.198,169.653,41.368,157.794
C08580=1036.344,137.593,-98.218,169.655,41.368,157.794
C08581=1036.350,137.842,-98.240,169.657,41.368,157.794
C08582=1036.356,138.092,-98.262,169.660,41.368,157.794
C08583=1036.362,138.340,-98.283,169.662,41.368,157.794
C08584=1036.369,138.589,-98.304,169.665,41.367,157.794
C08585=1036.375,138.839,-98.325,169.667,41.367,157.794
C08586=1036.381,139.088,-98.346,169.669,41.367,157.794
C08587=1036.386,139.336,-98.368,169.672,41.367,157.794
C08588=1036.392,139.586,-98.389,169.674,41.366,157.794
C08589=1036.399,139.835,-98.410,169.676,41.366,157.795
C08590=1036.405,140.083,-98.432,169.679,41.366,157.795
C08591=1036.411,140.332,-98.453,169.681,41.365,157.795
C08592=1036.418,140.617,-98.478,169.685,41.366,157.795
C08593=1036.425,140.903,-98.502,169.688,41.365,157.795
C08594=1036.432,141.189,-98.527,169.690,41.365,157.795
C08595=1036.438,141.474,-98.552,169.693,41.365,157.795
C08596=1036.445,141.723,-98.574,169.695,41.364,157.795
C08597=1036.451,141.972,-98.595,169.698,41.364,157.795
C08598=1036.458,142.221,-98.617,169.700,41.364,157.796
C08599=1036.464,142.470,-98.638,169.703,41.364,157.796
C08600=1036.469,142.719,-98.659,169.705,41.364,157.796
C08601=1036.476,142.968,-98.681,169.707,41.363,157.796
C08602=1036.482,143.217,-98.703,169.710,41.363,157.796
C08603=1036.488,143.466,-98.724,169.712,41.363,157.796
C08604=1036.493,143.715,-98.746,169.715,41.362,157.796
C08605=1036.500,143.964,-98.767,169.717,41.363,157.796
C08606=1036.506,144.213,-98.789,169.719,41.363,157.796
C08607=1036.512,144.462,-98.810,169.722,41.362,157.796
C08608=1036.518,144.712,-98.832,169.724,41.362,157.796
C08609=1036.524,144.960,-98.853,169.727,41.362,157.796
C08610=1036.531,145.209,-98.874,169.729,41.361,157.797
C08611=1036.537,145.458,-98.896,169.731,41.361,157.797
C08612=1036.543,145.707,-98.918,169.734,41.361,157.797
C08613=1036.549,145.956,-98.940,169.737,41.361,157.797
C08614=1036.555,146.205,-98.962,169.740,41.361,157.797
C08615=1036.562,146.454,-98.983,169.742,41.360,157.797
C08616=1036.567,146.703,-99.005,169.745,41.360,157.797
C08617=1036.573,146.952,-99.026,169.747,41.360,157.797
C08618=1036.580,147.201,-99.049,169.749,41.359,157.797
C08619=1036.586,147.450,-99.070,169.752,41.360,157.798
C08620=1036.592,147.699,-99.092,169.754,41.359,157.798
C08621=1036.598,147.948,-99.113,169.757,41.359,157.798
C08622=1036.604,148.196,-99.135,169.759,41.359,157.798
C08623=1036.610,148.446,-99.158,169.761,41.359,157.798
C08624=1036.616,148.695,-99.179,169.764,41.359,157.798
C08625=1036.622,148.944,-99.201,169.766,41.359,157.798
C08626=1036.628,149.193,-99.223,169.769,41.358,157.798
C08627=1036.635,149.442,-99.245,169.771,41.358,157.798
C08628=1036.641,149.691,-99.267,169.775,41.358,157.798
C08629=1036.647,149.940,-99.289,169.777,41.358,157.799
C08630=1036.652,150.189,-99.311,169.779,41.358,157.799
C08631=1036.658,150.438,-99.332,169.782,41.357,157.799
C08632=1036.665,150.686,-99.355,169.784,41.358,157.799
C08633=1036.671,150.936,-99.376,169.787,41.357,157.799
C08634=1036.677,151.185,-99.398,169.789,41.357,157.799
C08635=1036.683,151.433,-99.420,169.792,41.357,157.799
C08636=1036.689,151.683,-99.443,169.794,41.357,157.799
C08637=1036.695,151.931,-99.465,169.796,41.357,157.799
C08638=1036.702,152.181,-99.487,169.799,41.356,157.799
C08639=1036.708,152.430,-99.508,169.801,41.357,157.800
C08640=1036.714,152.678,-99.530,169.804,41.356,157.800
C08641=1036.719,152.927,-99.552,169.806,41.356,157.800
C08642=1036.725,153.176,-99.575,169.810,41.356,157.800
C08643=1036.732,153.425,-99.596,169.812,41.356,157.800
C08644=1036.738,153.674,-99.619,169.815,41.356,157.800
C08645=1036.744,153.923,-99.640,169.817,41.355,157.800
C08646=1036.750,154.172,-99.663,169.820,41.355,157.800
C08647=1036.756,154.421,-99.685,169.822,41.355,157.801
C08648=1036.763,154.669,-99.707,169.825,41.355,157.801
C08649=1036.768,154.919,-99.730,169.827,41.355,157.801
C08650=1036.775,155.168,-99.752,169.829,41.355,157.801
C08651=1036.781,155.417,-99.774,169.832,41.355,157.801
C08652=1036.786,155.666,-99.797,169.834,41.355,157.801
C08653=1036.793,155.914,-99.819,169.838,41.355,157.801
C08654=1036.799,156.163,-99.841,169.840,41.355,157.801
C08655=1036.805,156.412,-99.863,169.843,41.354,157.801
C08656=1036.811,156.697,-99.888,169.846,41.354,157.802
C08657=1036.819,156.983,-99.915,169.848,41.354,157.802
C08658=1036.825,157.268,-99.939,169.851,41.354,157.802
C08659=1036.833,157.553,-99.966,169.854,41.354,157.802
C08660=1036.839,157.802,-99.987,169.857,41.354,157.802
C08661=1036.846,158.051,-100.009,169.859,41.354,157.802
C08662=1036.851,158.300,-100.032,169.862,41.354,157.802
C08663=1036.857,158.549,-100.054,169.864,41.353,157.803
C08664=1036.864,158.797,-100.076,169.868,41.354,157.803
C08665=1036.870,159.046,-100.099,169.870,41.353,157.803
C08666=1036.876,159.295,-100.121,169.873,41.353,157.803
C08667=1036.881,159.544,-100.144,169.875,41.353,157.803
C08668=1036.888,159.793,-100.166,169.878,41.353,157.803
C08669=1036.894,160.042,-100.189,169.880,41.353,157.803
C08670=1036.900,160.291,-100.211,169.883,41.353,157.803
C08671=1036.906,160.540,-100.234,169.885,41.353,157.804
C08672=1036.911,160.789,-100.257,169.887,41.353,157.804
C08673=1036.918,161.037,-100.279,169.890,41.353,157.804
C08674=1036.924,161.286,-100.302,169.893,41.353,157.804
C08675=1036.929,161.535,-100.325,169.896,41.353,157.804
C08676=1036.935,161.784,-100.348,169.898,41.353,157.804
C08677=1036.941,162.033,-100.371,169.901,41.353,157.805
C08678=1036.947,162.282,-100.393,169.903,41.354,157.805
C08679=1036.953,162.531,-100.415,169.906,41.353,157.805
C08680=1036.958,162.780,-100.438,169.908,41.354,157.805
C08681=1036.964,163.029,-100.461,169.911,41.353,157.805
C08682=1036.971,163.277,-100.484,169.914,41.354,157.805
C08683=1036.976,163.526,-100.507,169.917,41.353,157.805
C08684=1036.982,163.775,-100.530,169.919,41.354,157.806
C08685=1036.988,164.025,-100.553,169.922,41.354,157.806
C08686=1036.995,164.273,-100.575,169.924,41.354,157.806
C08687=1037.001,164.522,-100.598,169.927,41.354,157.806
C08688=1037.006,164.771,-100.621,169.929,41.354,157.806
C08689=1037.012,165.020,-100.644,169.932,41.354,157.806
C08690=1037.018,165.269,-100.667,169.935,41.354,157.807
C08691=1037.024,165.518,-100.689,169.938,41.354,157.807
C08692=1037.030,165.767,-100.712,169.940,41.354,157.807
C08693=1037.036,166.015,-100.735,169.943,41.354,157.807
C08694=1037.041,166.264,-100.758,169.945,41.354,157.807
C08695=1037.047,166.513,-100.781,169.948,41.354,157.807
C08696=1037.054,166.763,-100.804,169.950,41.354,157.807
C08697=1037.060,167.011,-100.828,169.954,41.355,157.808
C08698=1037.066,167.260,-100.851,169.956,41.354,157.808
C08699=1037.072,167.509,-100.873,169.959,41.355,157.808
C08700=1037.077,167.757,-100.896,169.961,41.354,157.808
C08701=1037.084,168.006,-100.919,169.964,41.355,157.808
C08702=1037.090,168.255,-100.942,169.967,41.355,157.809
C08703=1037.096,168.505,-100.965,169.969,41.355,157.809
C08704=1037.102,168.753,-100.988,169.972,41.355,157.809
C08705=1037.108,169.002,-101.012,169.974,41.355,157.809
C08706=1037.114,169.250,-101.034,169.978,41.355,157.809
C08707=1037.120,169.499,-101.057,169.980,41.355,157.809
C08708=1037.126,169.749,-101.080,169.983,41.355,157.809
C08709=1037.132,169.998,-101.103,169.985,41.355,157.810
C08710=1037.138,170.246,-101.127,169.988,41.355,157.810
C08711=1037.144,170.495,-101.150,169.991,41.355,157.810
C08712=1037.150,170.743,-101.172,169.994,41.355,157.810
C08713=1037.157,170.993,-101.195,169.997,41.355,157.810
C08714=1037.162,171.242,-101.218,169.999,41.355,157.810
C08715=1037.168,171.490,-101.242,170.002,41.355,157.810
C08716=1037.174,171.739,-101.265,170.004,41.355,157.811
C08717=1037.180,171.989,-101.288,170.007,41.356,157.811
C08718=1037.187,172.237,-101.311,170.010,41.355,157.811
C08719=1037.193,172.486,-101.334,170.012,41.356,157.811
C08720=1037.200,172.771,-101.361,170.016,41.356,157.811
C08721=1037.207,173.055,-101.387,170.019,41.356,157.812
C08722=1037.214,173.340,-101.414,170.022,41.356,157.812
C08723=1037.221,173.624,-101.440,170.025,41.356,157.812
C08724=1037.226,173.873,-101.463,170.028,41.356,157.812
C08725=1037.233,174.122,-101.487,170.030,41.356,157.812
C08726=1037.239,174.371,-101.510,170.034,41.356,157.812
C08727=1037.245,174.620,-101.533,170.037,41.356,157.813
C08728=1037.252,174.869,-101.557,170.039,41.356,157.813
C08729=1037.258,175.117,-101.580,170.042,41.356,157.813
C08730=1037.263,175.366,-101.603,170.045,41.356,157.813
C08731=1037.270,175.615,-101.627,170.047,41.357,157.813
C08732=1037.276,175.864,-101.650,170.050,41.356,157.813
C08733=1037.282,176.112,-101.673,170.053,41.356,157.814
C08734=1037.289,176.362,-101.696,170.056,41.357,157.814
C08735=1037.295,176.610,-101.720,170.059,41.356,157.814
C08736=1037.301,176.859,-101.743,170.061,41.357,157.814
C08737=1037.307,177.109,-101.766,170.064,41.357,157.814
C08738=1037.313,177.357,-101.790,170.067,41.357,157.814
C08739=1037.319,177.606,-101.813,170.069,41.357,157.815
C08740=1037.325,177.855,-101.837,170.072,41.357,157.815
C08741=1037.331,178.104,-101.859,170.076,41.357,157.815
C08742=1037.339,178.352,-101.883,170.078,41.357,157.815
C08743=1037.344,178.601,-101.906,170.081,41.357,157.815
C08744=1037.351,178.850,-101.930,170.084,41.357,157.815
C08745=1037.357,179.098,-101.954,170.087,41.357,157.816
C08746=1037.363,179.347,-101.976,170.089,41.357,157.816
C08747=1037.369,179.596,-102.001,170.092,41.357,157.816
C08748=1037.375,179.845,-102.023,170.096,41.358,157.816
C08749=1037.382,180.094,-102.047,170.098,41.357,157.816
C08750=1037.388,180.343,-102.070,170.101,41.358,157.816
C08751=1037.395,180.592,-102.094,170.104,41.358,157.817
C08752=1037.401,180.840,-102.118,170.106,41.358,157.817
C08753=1037.407,181.090,-102.141,170.109,41.358,157.817
C08754=1037.413,181.338,-102.164,170.112,41.358,157.817
C08755=1037.419,181.587,-102.188,170.116,41.358,157.817
C08756=1037.426,181.836,-102.211,170.118,41.358,157.818
C08757=1037.432,182.085,-102.235,170.121,41.358,157.818
C08758=1037.438,182.334,-102.258,170.124,41.359,157.818
C08759=1037.445,182.583,-102.282,170.126,41.358,157.818
C08760=1037.451,182.831,-102.306,170.129,41.359,157.818
C08761=1037.458,183.080,-102.330,170.133,41.359,157.819
C08762=1037.464,183.328,-102.353,170.136,41.358,157.819
C08763=1037.470,183.578,-102.377,170.138,41.359,157.819
C08764=1037.476,183.826,-102.401,170.141,41.359,157.819
C08765=1037.481,184.075,-102.425,170.144,41.359,157.819
C08766=1037.488,184.324,-102.449,170.146,41.360,157.819
C08767=1037.494,184.572,-102.473,170.150,41.360,157.820
C08768=1037.500,184.821,-102.497,170.153,41.360,157.820
C08769=1037.505,185.070,-102.520,170.155,41.360,157.820
C08770=1037.511,185.319,-102.545,170.158,41.361,157.820
C08771=1037.517,185.568,-102.569,170.161,41.361,157.821
C08772=1037.523,185.817,-102.593,170.164,41.361,157.821
C08773=1037.529,186.065,-102.617,170.167,41.362,157.821
C08774=1037.534,186.314,-102.641,170.170,41.362,157.821
C08775=1037.541,186.563,-102.665,170.172,41.362,157.821
C08776=1037.546,186.811,-102.689,170.175,41.362,157.822
C08777=1037.553,187.060,-102.713,170.179,41.363,157.822
C08778=1037.558,187.309,-102.738,170.182,41.363,157.822
C08779=1037.565,187.558,-102.762,170.184,41.364,157.822
C08780=1037.570,187.806,-102.786,170.187,41.364,157.823
C08781=1037.577,188.055,-102.811,170.191,41.364,157.823
C08782=1037.582,188.303,-102.835,170.193,41.365,157.823
C08783=1037.589,188.552,-102.859,170.196,41.365,157.823
C08784=1037.596,188.837,-102.886,170.199,41.365,157.824
C08785=1037.603,189.121,-102.914,170.202,41.366,157.824
C08786=1037.610,189.406,-102.941,170.207,41.366,157.824
C08787=1037.617,189.689,-102.969,170.210,41.367,157.824
C08788=1037.623,189.938,-102.994,170.212,41.367,157.825
C08789=1037.629,190.187,-103.017,170.215,41.367,157.825
C08790=1037.635,190.436,-103.042,170.219,41.367,157.825
C08791=1037.641,190.684,-103.067,170.222,41.368,157.825
C08792=1037.647,190.933,-103.091,170.224,41.368,157.825
C08793=1037.653,191.182,-103.115,170.227,41.368,157.826
C08794=1037.659,191.430,-103.139,170.230,41.369,157.826
C08795=1037.665,191.679,-103.163,170.234,41.369,157.826
C08796=1037.672,191.928,-103.189,170.236,41.369,157.826
C08797=1037.678,192.176,-103.212,170.239,41.369,157.827
C08798=1037.684,192.426,-103.237,170.242,41.370,157.827
C08799=1037.689,192.675,-103.262,170.245,41.370,157.827
C08800=1037.696,192.923,-103.286,170.249,41.371,157.827
C08801=1037.702,193.172,-103.311,170.251,41.371,157.828
C08802=1037.708,193.421,-103.335,170.254,41.371,157.828
C08803=1037.714,193.669,-103.359,170.257,41.372,157.828
C08804=1037.721,193.918,-103.384,170.261,41.372,157.828
C08805=1037.726,194.167,-103.408,170.264,41.372,157.829
C08806=1037.732,194.415,-103.432,170.266,41.372,157.829
C08807=1037.739,194.664,-103.457,170.269,41.373,157.829
C08808=1037.745,194.913,-103.481,170.272,41.373,157.829
C08809=1037.751,195.162,-103.506,170.276,41.374,157.830
C08810=1037.758,195.410,-103.530,170.279,41.374,157.830
C08811=1037.763,195.659,-103.555,170.281,41.374,157.830
C08812=1037.770,195.908,-103.579,170.284,41.375,157.830
C08813=1037.776,196.156,-103.604,170.288,41.375,157.830
C08814=1037.782,196.405,-103.628,170.291,41.375,157.831
C08815=1037.789,196.654,-103.653,170.294,41.375,157.831
C08816=1037.794,196.903,-103.678,170.297,41.376,157.831
C08817=1037.801,197.151,-103.702,170.300,41.377,157.831
C08818=1037.807,197.400,-103.727,170.303,41.377,157.832
C08819=1037.813,197.649,-103.751,170.306,41.377,157.832
C08820=1037.820,197.898,-103.776,170.309,41.377,157.832
C08821=1037.826,198.146,-103.800,170.312,41.378,157.832
C08822=1037.832,198.395,-103.825,170.316,41.378,157.833
C08823=1037.838,198.644,-103.849,170.319,41.379,157.833
C08824=1037.845,198.931,-103.879,170.322,41.379,157.833
C08825=1037.853,199.217,-103.907,170.326,41.380,157.834
C08826=1037.860,199.504,-103.935,170.330,41.380,157.834
C08827=1037.867,199.790,-103.964,170.333,41.380,157.834
C08828=1037.874,200.039,-103.988,170.336,41.381,157.834
C08829=1037.880,200.288,-104.013,170.340,41.381,157.835
C08830=1037.886,200.537,-104.038,170.343,41.382,157.835
C08831=1037.893,200.786,-104.062,170.345,41.382,157.835
C08832=1037.899,201.034,-104.088,170.348,41.382,157.835
C08833=1037.905,201.283,-104.113,170.352,41.383,157.836
C08834=1037.910,201.532,-104.137,170.355,41.383,157.836
C08835=1037.916,201.780,-104.163,170.358,41.384,157.836
C08836=1037.923,202.029,-104.188,170.361,41.384,157.836
C08837=1037.930,202.277,-104.213,170.365,41.385,157.837
C08838=1037.935,202.527,-104.237,170.368,41.385,157.837
C08839=1037.942,202.775,-104.263,170.370,41.386,157.837
C08840=1037.947,203.023,-104.288,170.374,41.387,157.838
C08841=1037.953,203.272,-104.313,170.377,41.387,157.838
C08842=1037.960,203.520,-104.338,170.380,41.388,157.838
C08843=1037.966,203.770,-104.363,170.383,41.388,157.838
C08844=1037.972,204.006,-104.387,170.387,41.388,157.839
C08845=1037.977,204.243,-104.410,170.389,41.389,157.839
C08846=1037.983,204.479,-104.435,170.392,41.390,157.839
C08847=1038.013,205.663,-104.555,170.696,41.494,157.878
C08848=1038.021,205.981,-104.588,170.699,41.496,157.879
C08849=1038.030,206.299,-104.622,170.702,41.497,157.879
C08850=1038.039,206.617,-104.655,170.705,41.499,157.880
C08851=1038.048,206.935,-104.690,170.708,41.500,157.880
C08852=1038.054,207.183,-104.716,170.710,41.501,157.880
C08853=1038.061,207.432,-104.743,170.713,41.503,157.881
C08854=1038.067,207.680,-104.769,170.715,41.504,157.881
C08855=1038.074,207.929,-104.795,170.717,41.506,157.882
C08856=1038.081,208.178,-104.822,170.719,41.507,157.882
C08857=1038.087,208.426,-104.848,170.722,41.508,157.882
C08858=1038.094,208.675,-104.875,170.724,41.509,157.883
C08859=1038.101,208.924,-104.901,170.727,41.510,157.883
C08860=1038.108,209.171,-104.928,170.729,41.512,157.884
C08861=1038.115,209.420,-104.955,170.731,41.513,157.884
C08862=1038.120,209.668,-104.982,170.734,41.514,157.885
C08863=1038.128,209.917,-105.008,170.735,41.516,157.885
C08864=1038.135,210.166,-105.034,170.738,41.517,157.885
C08865=1038.140,210.414,-105.061,170.740,41.518,157.886
C08866=1038.148,210.662,-105.088,170.743,41.519,157.886
C08867=1038.155,210.911,-105.115,170.745,41.521,157.887
C08868=1038.161,211.159,-105.141,170.748,41.522,157.887
C08869=1038.168,211.408,-105.168,170.750,41.523,157.887
C08870=1038.175,211.657,-105.195,170.753,41.524,157.888
C08871=1038.181,211.905,-105.221,170.755,41.526,157.888
C08872=1038.187,212.154,-105.248,170.756,41.527,157.889
C08873=1038.195,212.403,-105.275,170.759,41.529,157.889
C08874=1038.201,212.650,-105.302,170.761,41.530,157.889
C08875=1038.208,212.899,-105.329,170.764,41.531,157.890
C08876=1038.214,213.148,-105.356,170.766,41.532,157.890
C08877=1038.221,213.395,-105.382,170.769,41.534,157.891
C08878=1038.227,213.645,-105.409,170.771,41.535,157.891
C08879=1038.235,213.893,-105.437,170.774,41.536,157.891
C08880=1038.241,214.141,-105.463,170.776,41.537,157.892
C08881=1038.248,214.390,-105.490,170.779,41.539,157.892
C08882=1038.254,214.638,-105.517,170.780,41.540,157.893
C08883=1038.261,214.886,-105.543,170.783,41.542,157.893
C08884=1038.267,215.135,-105.570,170.785,41.543,157.893
C08885=1038.274,215.384,-105.598,170.788,41.544,157.894
C08886=1038.281,215.633,-105.625,170.790,41.545,157.894
C08887=1038.287,215.880,-105.652,170.793,41.547,157.895
C08888=1038.294,216.129,-105.678,170.795,41.548,157.895
C08889=1038.301,216.377,-105.706,170.797,41.549,157.896
C08890=1038.308,216.626,-105.733,170.800,41.550,157.896
C08891=1038.314,216.874,-105.760,170.802,41.552,157.896
C08892=1038.321,217.123,-105.786,170.805,41.553,157.897
C08893=1038.328,217.371,-105.814,170.807,41.555,157.897
C08894=1038.334,217.620,-105.841,170.810,41.556,157.898
C08895=1038.341,217.868,-105.868,170.812,41.557,157.898
C08896=1038.347,218.117,-105.895,170.815,41.558,157.898
C08897=1038.355,218.365,-105.922,170.817,41.560,157.899
C08898=1038.361,218.614,-105.949,170.820,41.561,157.899
C08899=1038.369,218.862,-105.976,170.822,41.562,157.900
C08900=1038.374,219.110,-106.003,170.824,41.563,157.900
C08901=1038.381,219.359,-106.031,170.827,41.564,157.900
C08902=1038.388,219.608,-106.057,170.829,41.566,157.901
C08903=1038.395,219.856,-106.085,170.832,41.567,157.901
C08904=1038.404,220.180,-106.120,170.835,41.569,157.902
C08905=1038.412,220.503,-106.156,170.838,41.571,157.902
C08906=1038.421,220.827,-106.192,170.842,41.572,157.903
C08907=1038.429,221.151,-106.227,170.844,41.574,157.904
C08908=1038.436,221.399,-106.255,170.847,41.575,157.904
C08909=1038.443,221.648,-106.281,170.849,41.577,157.904
C08910=1038.450,221.896,-106.309,170.852,41.578,157.905
C08911=1038.456,222.145,-106.336,170.854,41.579,157.905
C08912=1038.462,222.392,-106.364,170.857,41.580,157.906
C08913=1038.469,222.641,-106.391,170.859,41.582,157.906
C08914=1038.475,222.890,-106.419,170.862,41.584,157.907
C08915=1038.482,223.138,-106.446,170.864,41.585,157.907
C08916=1038.490,223.386,-106.473,170.867,41.586,157.907
C08917=1038.496,223.635,-106.500,170.869,41.587,157.908
C08918=1038.503,223.884,-106.528,170.872,41.589,157.908
C08919=1038.509,224.132,-106.556,170.874,41.590,157.909
C08920=1038.515,224.380,-106.583,170.877,41.591,157.909
C08921=1038.522,224.629,-106.611,170.879,41.592,157.909
C08922=1038.529,224.877,-106.638,170.882,41.594,157.910
C08923=1038.536,225.126,-106.665,170.885,41.595,157.910
C08924=1038.542,225.374,-106.693,170.887,41.596,157.911
C08925=1038.549,225.623,-106.721,170.890,41.598,157.911
C08926=1038.556,225.871,-106.748,170.892,41.599,157.912
C08927=1038.563,226.119,-106.776,170.895,41.600,157.912
C08928=1038.569,226.367,-106.803,170.897,41.601,157.912
C08929=1038.576,226.615,-106.831,170.900,41.603,157.913
C08930=1038.583,226.864,-106.858,170.902,41.604,157.913
C08931=1038.589,227.112,-106.886,170.905,41.606,157.914
C08932=1038.596,227.361,-106.914,170.907,41.606,157.914
C08933=1038.602,227.610,-106.941,170.910,41.608,157.915
C08934=1038.609,227.858,-106.969,170.912,41.609,157.915
C08935=1038.616,228.107,-106.996,170.915,41.611,157.915
C08936=1038.623,228.355,-107.024,170.918,41.611,157.916
C08937=1038.629,228.604,-107.052,170.921,41.613,157.916
C08938=1038.636,228.852,-107.079,170.923,41.615,157.917
C08939=1038.643,229.100,-107.108,170.926,41.616,157.917
C08940=1038.650,229.348,-107.136,170.928,41.617,157.918
C08941=1038.656,229.597,-107.163,170.931,41.619,157.918
C08942=1038.663,229.845,-107.191,170.933,41.620,157.918
C08943=1038.670,230.094,-107.219,170.936,41.621,157.919
C08944=1038.676,230.342,-107.247,170.938,41.622,157.919
C08945=1038.683,230.590,-107.274,170.941,41.624,157.920
C08946=1038.690,230.839,-107.302,170.943,41.626,157.920
C08947=1038.696,231.087,-107.330,170.947,41.626,157.921
C08948=1038.703,231.335,-107.359,170.949,41.628,157.921
C08949=1038.709,231.584,-107.387,170.952,41.630,157.922
C08950=1038.716,231.832,-107.414,170.954,41.630,157.922
C08951=1038.723,232.081,-107.442,170.957,41.632,157.922
C08952=1038.729,232.329,-107.470,170.959,41.633,157.923
C08953=1038.736,232.577,-107.498,170.962,41.635,157.923
C08954=1038.742,232.826,-107.526,170.964,41.636,157.924
C08955=1038.749,233.074,-107.554,170.967,41.638,157.924
C08956=1038.756,233.323,-107.582,170.970,41.639,157.925
C08957=1038.763,233.570,-107.610,170.973,41.640,157.925
C08958=1038.769,233.819,-107.639,170.975,41.642,157.926
C08959=1038.775,234.068,-107.666,170.978,41.643,157.926
C08960=1038.785,234.450,-107.710,170.981,41.645,157.927
C08961=1038.796,234.832,-107.753,170.986,41.647,157.927
C08962=1038.806,235.214,-107.797,170.990,41.649,157.928
C08963=1038.816,235.597,-107.840,170.994,41.652,157.929
C08964=1038.823,235.846,-107.868,170.996,41.652,157.929
C08965=1038.830,236.094,-107.896,171.000,41.654,157.930
C08966=1038.836,236.342,-107.925,171.002,41.656,157.930
C08967=1038.843,236.590,-107.953,171.005,41.656,157.930
C08968=1038.849,236.839,-107.981,171.007,41.658,157.931
C08969=1038.856,237.087,-108.009,171.010,41.660,157.931
C08970=1038.862,237.335,-108.038,171.012,41.661,157.932
C08971=1038.869,237.584,-108.065,171.016,41.662,157.932
C08972=1038.875,237.799,-108.090,171.018,41.663,157.933
C08973=1038.882,238.014,-108.115,171.020,41.665,157.933
C08974=1038.886,238.229,-108.139,171.022,41.666,157.933
C08975=1038.892,238.445,-108.163,171.025,41.667,157.934
C08976=1038.898,238.659,-108.188,171.027,41.668,157.934
C08977=1038.904,238.875,-108.213,171.029,41.669,157.935
C08978=1038.910,239.091,-108.237,171.032,41.670,157.935
C08979=1038.916,239.305,-108.262,171.034,41.672,157.935
C08980=1038.923,239.554,-108.290,171.037,41.673,157.936
C08981=1038.929,239.802,-108.319,171.039,41.674,157.936
C08982=1038.936,240.050,-108.347,171.043,41.676,157.937
C08983=1038.942,240.299,-108.376,171.045,41.677,157.937
C08984=1038.949,240.546,-108.404,171.048,41.678,157.938
C08985=1038.956,240.795,-108.432,171.050,41.680,157.938
C08986=1038.963,241.044,-108.461,171.054,41.681,157.938
C08987=1038.969,241.292,-108.489,171.056,41.682,157.939
C08988=1038.976,241.540,-108.518,171.059,41.684,157.939
C08989=1038.983,241.788,-108.547,171.062,41.685,157.940
C08990=1038.989,242.036,-108.576,171.064,41.686,157.940
C08991=1038.995,242.285,-108.604,171.067,41.688,157.941
C08992=1039.002,242.534,-108.633,171.070,41.689,157.941
C08993=1039.009,242.782,-108.662,171.073,41.691,157.942
C08994=1039.016,243.029,-108.690,171.075,41.693,157.942
C08995=1039.021,243.278,-108.719,171.079,41.693,157.943
C08996=1039.028,243.526,-108.747,171.081,41.695,157.943
C08997=1039.035,243.774,-108.776,171.084,41.697,157.944
C08998=1039.042,244.023,-108.806,171.086,41.698,157.944
C08999=1039.049,244.271,-108.834,171.090,41.700,157.945
C09000=1039.054,244.520,-108.862,171.092,41.700,157.945
C09001=1039.061,244.767,-108.891,171.095,41.702,157.946
C09002=1039.068,245.016,-108.920,171.097,41.704,157.946
C09003=1039.075,245.264,-108.949,171.101,41.705,157.947
C09004=1039.081,245.513,-108.978,171.104,41.707,157.947
C09005=1039.088,245.760,-109.007,171.106,41.708,157.948
C09006=1039.094,246.008,-109.036,171.109,41.710,157.948
C09007=1039.101,246.257,-109.065,171.112,41.711,157.948
C09008=1039.107,246.505,-109.094,171.115,41.712,157.949
C09009=1039.113,246.754,-109.123,171.117,41.714,157.949
C09010=1039.120,247.002,-109.152,171.120,41.715,157.950
C09011=1039.127,247.249,-109.181,171.123,41.717,157.950
C09012=1039.133,247.498,-109.210,171.126,41.718,157.951
C09013=1039.140,247.746,-109.239,171.128,41.720,157.951
C09014=1039.146,247.995,-109.268,171.132,41.721,157.952
C09015=1039.152,248.243,-109.297,171.135,41.723,157.952
C09016=1039.161,248.553,-109.334,171.138,41.724,157.953
C09017=1039.169,248.864,-109.370,171.142,41.726,157.954
